   1:  PR[GP1:91,1] = PR[GP1:90,1] + -1.924;
   1:  PR[GP1:91,2] = PR[GP1:90,2] + -33.395;
   1:L PR[91] 10mm/sec CNT100;
   1:  PR[GP1:91,1] = PR[GP1:90,1] + -0.973;
   1:  PR[GP1:91,2] = PR[GP1:90,2] + -33.399;
   1:L PR[91] 10mm/sec CNT100;
   1:  PR[GP1:91,1] = PR[GP1:90,1] + 1.461;
   1:  PR[GP1:91,2] = PR[GP1:90,2] + -33.302;
   1:L PR[91] 10mm/sec CNT100;
   1:  PR[GP1:91,1] = PR[GP1:90,1] + 2.467;
   1:  PR[GP1:91,2] = PR[GP1:90,2] + -33.088;
   1:L PR[91] 10mm/sec CNT100;
   1:  PR[GP1:91,1] = PR[GP1:90,1] + 2.933;
   1:  PR[GP1:91,2] = PR[GP1:90,2] + -33.462;
   1:L PR[91] 10mm/sec CNT100;
   1:  PR[GP1:91,1] = PR[GP1:90,1] + 7.580;
   1:  PR[GP1:91,2] = PR[GP1:90,2] + -34.974;
   1:L PR[91] 10mm/sec CNT100;
   1:  PR[GP1:91,1] = PR[GP1:90,1] + 15.667;
   1:  PR[GP1:91,2] = PR[GP1:90,2] + -37.774;
   1:L PR[91] 10mm/sec CNT100;
   1:  PR[GP1:91,1] = PR[GP1:90,1] + 15.934;
   1:  PR[GP1:91,2] = PR[GP1:90,2] + -37.809;
   1:L PR[91] 10mm/sec CNT100;
   1:  PR[GP1:91,1] = PR[GP1:90,1] + 16.325;
   1:  PR[GP1:91,2] = PR[GP1:90,2] + -37.796;
   1:L PR[91] 10mm/sec CNT100;
   1:  PR[GP1:91,1] = PR[GP1:90,1] + 29.643;
   1:  PR[GP1:91,2] = PR[GP1:90,2] + -37.737;
   1:L PR[91] 10mm/sec CNT100;
   1:  PR[GP1:91,1] = PR[GP1:90,1] + 30.537;
   1:  PR[GP1:91,2] = PR[GP1:90,2] + -37.545;
   1:L PR[91] 10mm/sec CNT100;
   1:  PR[GP1:91,1] = PR[GP1:90,1] + 31.585;
   1:  PR[GP1:91,2] = PR[GP1:90,2] + -37.132;
   1:L PR[91] 10mm/sec CNT100;
   1:  PR[GP1:91,1] = PR[GP1:90,1] + 42.786;
   1:  PR[GP1:91,2] = PR[GP1:90,2] + -33.162;
   1:L PR[91] 10mm/sec CNT100;
   1:  PR[GP1:91,1] = PR[GP1:90,1] + 44.099;
   1:  PR[GP1:91,2] = PR[GP1:90,2] + -32.349;
   1:L PR[91] 10mm/sec CNT100;
   1:  PR[GP1:91,1] = PR[GP1:90,1] + 45.422;
   1:  PR[GP1:91,2] = PR[GP1:90,2] + -31.177;
   1:L PR[91] 10mm/sec CNT100;
   1:  PR[GP1:91,1] = PR[GP1:90,1] + 53.505;
   1:  PR[GP1:91,2] = PR[GP1:90,2] + -24.634;
   1:L PR[91] 10mm/sec CNT100;
   1:  PR[GP1:91,1] = PR[GP1:90,1] + 54.760;
   1:  PR[GP1:91,2] = PR[GP1:90,2] + -23.005;
   1:L PR[91] 10mm/sec CNT100;
   1:  PR[GP1:91,1] = PR[GP1:90,1] + 55.835;
   1:  PR[GP1:91,2] = PR[GP1:90,2] + -20.942;
   1:L PR[91] 10mm/sec CNT100;
   1:  PR[GP1:91,1] = PR[GP1:90,1] + 60.576;
   1:  PR[GP1:91,2] = PR[GP1:90,2] + -13.042;
   1:L PR[91] 10mm/sec CNT100;
   1:  PR[GP1:91,1] = PR[GP1:90,1] + 61.225;
   1:  PR[GP1:91,2] = PR[GP1:90,2] + -10.871;
   1:L PR[91] 10mm/sec CNT100;
   1:  PR[GP1:91,1] = PR[GP1:90,1] + 61.456;
   1:  PR[GP1:91,2] = PR[GP1:90,2] + -8.401;
   1:L PR[91] 10mm/sec CNT100;
   1:  PR[GP1:91,1] = PR[GP1:90,1] + 63.007;
   1:  PR[GP1:91,2] = PR[GP1:90,2] + 0.023;
   1:L PR[91] 10mm/sec CNT100;
   1:  PR[GP1:91,1] = PR[GP1:90,1] + 62.779;
   1:  PR[GP1:91,2] = PR[GP1:90,2] + 2.498;
   1:L PR[91] 10mm/sec CNT100;
   1:  PR[GP1:91,1] = PR[GP1:90,1] + 61.234;
   1:  PR[GP1:91,2] = PR[GP1:90,2] + 10.834;
   1:L PR[91] 10mm/sec CNT100;
   1:  PR[GP1:91,1] = PR[GP1:90,1] + 60.572;
   1:  PR[GP1:91,2] = PR[GP1:90,2] + 13.050;
   1:L PR[91] 10mm/sec CNT100;
   1:  PR[GP1:91,1] = PR[GP1:90,1] + 59.492;
   1:  PR[GP1:91,2] = PR[GP1:90,2] + 15.141;
   1:L PR[91] 10mm/sec CNT100;
   1:  PR[GP1:91,1] = PR[GP1:90,1] + 54.775;
   1:  PR[GP1:91,2] = PR[GP1:90,2] + 22.977;
   1:L PR[91] 10mm/sec CNT100;
   1:  PR[GP1:91,1] = PR[GP1:90,1] + 53.500;
   1:  PR[GP1:91,2] = PR[GP1:90,2] + 24.633;
   1:L PR[91] 10mm/sec CNT100;
   1:  PR[GP1:91,1] = PR[GP1:90,1] + 52.084;
   1:  PR[GP1:91,2] = PR[GP1:90,2] + 25.898;
   1:L PR[91] 10mm/sec CNT100;
   1:  PR[GP1:91,1] = PR[GP1:90,1] + 44.120;
   1:  PR[GP1:91,2] = PR[GP1:90,2] + 32.328;
   1:L PR[91] 10mm/sec CNT100;
   1:  PR[GP1:91,1] = PR[GP1:90,1] + 42.785;
   1:  PR[GP1:91,2] = PR[GP1:90,2] + 33.155;
   1:L PR[91] 10mm/sec CNT100;
   1:  PR[GP1:91,1] = PR[GP1:90,1] + 41.460;
   1:  PR[GP1:91,2] = PR[GP1:90,2] + 33.684;
   1:L PR[91] 10mm/sec CNT100;
   1:  PR[GP1:91,1] = PR[GP1:90,1] + 30.563;
   1:  PR[GP1:91,2] = PR[GP1:90,2] + 37.531;
   1:L PR[91] 10mm/sec CNT100;
   1:  PR[GP1:91,1] = PR[GP1:90,1] + 29.649;
   1:  PR[GP1:91,2] = PR[GP1:90,2] + 37.728;
   1:L PR[91] 10mm/sec CNT100;
   1:  PR[GP1:91,1] = PR[GP1:90,1] + 28.809;
   1:  PR[GP1:91,2] = PR[GP1:90,2] + 37.760;
   1:L PR[91] 10mm/sec CNT100;
   1:  PR[GP1:91,1] = PR[GP1:90,1] + 15.964;
   1:  PR[GP1:91,2] = PR[GP1:90,2] + 37.805;
   1:L PR[91] 10mm/sec CNT100;
   1:  PR[GP1:91,1] = PR[GP1:90,1] + 15.687;
   1:  PR[GP1:91,2] = PR[GP1:90,2] + 37.768;
   1:L PR[91] 10mm/sec CNT100;
   1:  PR[GP1:91,1] = PR[GP1:90,1] + 7.446;
   1:  PR[GP1:91,2] = PR[GP1:90,2] + 34.920;
   1:L PR[91] 10mm/sec CNT100;
   1:  PR[GP1:91,1] = PR[GP1:90,1] + 3.248;
   1:  PR[GP1:91,2] = PR[GP1:90,2] + 33.556;
   1:L PR[91] 10mm/sec CNT100;
   1:  PR[GP1:91,1] = PR[GP1:90,1] + 2.438;
   1:  PR[GP1:91,2] = PR[GP1:90,2] + 33.105;
   1:L PR[91] 10mm/sec CNT100;
   1:  PR[GP1:91,1] = PR[GP1:90,1] + 0.251;
   1:  PR[GP1:91,2] = PR[GP1:90,2] + 33.820;
   1:  PR[GP1:91,3] = PR[GP1:90,3] + 71.820;
   1:L PR[91] 10mm/sec CNT100;
   1:  PR[GP1:91,1] = PR[GP1:90,1] + -1.865;
   1:  PR[GP1:91,2] = PR[GP1:90,2] + 33.807;
   1:L PR[91] 10mm/sec CNT100;
   1:  PR[GP1:91,1] = PR[GP1:90,1] + -14.438;
   1:  PR[GP1:91,2] = PR[GP1:90,2] + 37.919;
   1:L PR[91] 10mm/sec CNT100;
   1:  PR[GP1:91,1] = PR[GP1:90,1] + -28.437;
   1:  PR[GP1:91,2] = PR[GP1:90,2] + 37.848;
   1:L PR[91] 10mm/sec CNT100;
   1:  PR[GP1:91,1] = PR[GP1:90,1] + -28.988;
   1:  PR[GP1:91,2] = PR[GP1:90,2] + 37.729;
   1:L PR[91] 10mm/sec CNT100;
   1:  PR[GP1:91,1] = PR[GP1:90,1] + -29.665;
   1:  PR[GP1:91,2] = PR[GP1:90,2] + 37.461;
   1:L PR[91] 10mm/sec CNT100;
   1:  PR[GP1:91,1] = PR[GP1:90,1] + -41.584;
   1:  PR[GP1:91,2] = PR[GP1:90,2] + 33.229;
   1:L PR[91] 10mm/sec CNT100;
   1:  PR[GP1:91,1] = PR[GP1:90,1] + -42.596;
   1:  PR[GP1:91,2] = PR[GP1:90,2] + 32.598;
   1:L PR[91] 10mm/sec CNT100;
   1:  PR[GP1:91,1] = PR[GP1:90,1] + -43.632;
   1:  PR[GP1:91,2] = PR[GP1:90,2] + 31.678;
   1:L PR[91] 10mm/sec CNT100;
   1:  PR[GP1:91,1] = PR[GP1:90,1] + -52.315;
   1:  PR[GP1:91,2] = PR[GP1:90,2] + 24.651;
   1:L PR[91] 10mm/sec CNT100;
   1:  PR[GP1:91,1] = PR[GP1:90,1] + -53.335;
   1:  PR[GP1:91,2] = PR[GP1:90,2] + 23.323;
   1:L PR[91] 10mm/sec CNT100;
   1:  PR[GP1:91,1] = PR[GP1:90,1] + -54.225;
   1:  PR[GP1:91,2] = PR[GP1:90,2] + 21.596;
   1:L PR[91] 10mm/sec CNT100;
   1:  PR[GP1:91,1] = PR[GP1:90,1] + -59.359;
   1:  PR[GP1:91,2] = PR[GP1:90,2] + 13.022;
   1:L PR[91] 10mm/sec CNT100;
   1:  PR[GP1:91,1] = PR[GP1:90,1] + -59.908;
   1:  PR[GP1:91,2] = PR[GP1:90,2] + 11.157;
   1:L PR[91] 10mm/sec CNT100;
   1:  PR[GP1:91,1] = PR[GP1:90,1] + -60.096;
   1:  PR[GP1:91,2] = PR[GP1:90,2] + 9.107;
   1:L PR[91] 10mm/sec CNT100;
   1:  PR[GP1:91,1] = PR[GP1:90,1] + -61.780;
   1:  PR[GP1:91,2] = PR[GP1:90,2] + -0.032;
   1:L PR[91] 10mm/sec CNT100;
   1:  PR[GP1:91,1] = PR[GP1:90,1] + -61.594;
   1:  PR[GP1:91,2] = PR[GP1:90,2] + -2.098;
   1:L PR[91] 10mm/sec CNT100;
   1:  PR[GP1:91,1] = PR[GP1:90,1] + -59.915;
   1:  PR[GP1:91,2] = PR[GP1:90,2] + -11.142;
   1:L PR[91] 10mm/sec CNT100;
   1:  PR[GP1:91,1] = PR[GP1:90,1] + -59.352;
   1:  PR[GP1:91,2] = PR[GP1:90,2] + -13.053;
   1:L PR[91] 10mm/sec CNT100;
   1:  PR[GP1:91,1] = PR[GP1:90,1] + -58.438;
   1:  PR[GP1:91,2] = PR[GP1:90,2] + -14.845;
   1:L PR[91] 10mm/sec CNT100;
   1:  PR[GP1:91,1] = PR[GP1:90,1] + -53.343;
   1:  PR[GP1:91,2] = PR[GP1:90,2] + -23.322;
   1:L PR[91] 10mm/sec CNT100;
   1:  PR[GP1:91,1] = PR[GP1:90,1] + -52.301;
   1:  PR[GP1:91,2] = PR[GP1:90,2] + -24.678;
   1:L PR[91] 10mm/sec CNT100;
   1:  PR[GP1:91,1] = PR[GP1:90,1] + -51.126;
   1:  PR[GP1:91,2] = PR[GP1:90,2] + -25.732;
   1:L PR[91] 10mm/sec CNT100;
   1:  PR[GP1:91,1] = PR[GP1:90,1] + -42.599;
   1:  PR[GP1:91,2] = PR[GP1:90,2] + -32.605;
   1:L PR[91] 10mm/sec CNT100;
   1:  PR[GP1:91,1] = PR[GP1:90,1] + -41.563;
   1:  PR[GP1:91,2] = PR[GP1:90,2] + -33.250;
   1:L PR[91] 10mm/sec CNT100;
   1:  PR[GP1:91,1] = PR[GP1:90,1] + -40.542;
   1:  PR[GP1:91,2] = PR[GP1:90,2] + -33.660;
   1:L PR[91] 10mm/sec CNT100;
   1:  PR[GP1:91,1] = PR[GP1:90,1] + -28.983;
   1:  PR[GP1:91,2] = PR[GP1:90,2] + -37.738;
   1:L PR[91] 10mm/sec CNT100;
   1:  PR[GP1:91,1] = PR[GP1:90,1] + -28.411;
   1:  PR[GP1:91,2] = PR[GP1:90,2] + -37.862;
   1:L PR[91] 10mm/sec CNT100;
   1:  PR[GP1:91,1] = PR[GP1:90,1] + -27.878;
   1:  PR[GP1:91,2] = PR[GP1:90,2] + -37.882;
   1:L PR[91] 10mm/sec CNT100;
   1:  PR[GP1:91,1] = PR[GP1:90,1] + -14.415;
   1:  PR[GP1:91,2] = PR[GP1:90,2] + -37.925;
   1:L PR[91] 10mm/sec CNT100;
   1:  PR[GP1:91,1] = PR[GP1:90,1] + -1.865;
   1:  PR[GP1:91,2] = PR[GP1:90,2] + -33.819;
   1:L PR[91] 10mm/sec CNT100;
   1:  PR[GP1:91,1] = PR[GP1:90,1] + 0.338;
   1:  PR[GP1:91,2] = PR[GP1:90,2] + -33.830;
   1:L PR[91] 10mm/sec CNT100;
   1:  PR[GP1:91,1] = PR[GP1:90,1] + 1.823;
   1:  PR[GP1:91,2] = PR[GP1:90,2] + -33.770;
   1:L PR[91] 10mm/sec CNT100;
   1:  PR[GP1:91,1] = PR[GP1:90,1] + 2.534;
   1:  PR[GP1:91,2] = PR[GP1:90,2] + -33.619;
   1:L PR[91] 10mm/sec CNT100;
   1:  PR[GP1:91,1] = PR[GP1:90,1] + 2.874;
   1:  PR[GP1:91,2] = PR[GP1:90,2] + -33.893;
   1:L PR[91] 10mm/sec CNT100;
   1:  PR[GP1:91,1] = PR[GP1:90,1] + 14.365;
   1:  PR[GP1:91,2] = PR[GP1:90,2] + -37.631;
   1:L PR[91] 10mm/sec CNT100;
   1:  PR[GP1:91,1] = PR[GP1:90,1] + 15.195;
   1:  PR[GP1:91,2] = PR[GP1:90,2] + -37.918;
   1:L PR[91] 10mm/sec CNT100;
   1:  PR[GP1:91,1] = PR[GP1:90,1] + 29.235;
   1:  PR[GP1:91,2] = PR[GP1:90,2] + -37.861;
   1:L PR[91] 10mm/sec CNT100;
   1:  PR[GP1:91,1] = PR[GP1:90,1] + 29.785;
   1:  PR[GP1:91,2] = PR[GP1:90,2] + -37.742;
   1:L PR[91] 10mm/sec CNT100;
   1:  PR[GP1:91,1] = PR[GP1:90,1] + 30.462;
   1:  PR[GP1:91,2] = PR[GP1:90,2] + -37.476;
   1:L PR[91] 10mm/sec CNT100;
   1:  PR[GP1:91,1] = PR[GP1:90,1] + 42.388;
   1:  PR[GP1:91,2] = PR[GP1:90,2] + -33.249;
   1:L PR[91] 10mm/sec CNT100;
   1:  PR[GP1:91,1] = PR[GP1:90,1] + 43.393;
   1:  PR[GP1:91,2] = PR[GP1:90,2] + -32.626;
   1:L PR[91] 10mm/sec CNT100;
   1:  PR[GP1:91,1] = PR[GP1:90,1] + 44.423;
   1:  PR[GP1:91,2] = PR[GP1:90,2] + -31.714;
   1:L PR[91] 10mm/sec CNT100;
   1:  PR[GP1:91,1] = PR[GP1:90,1] + 53.109;
   1:  PR[GP1:91,2] = PR[GP1:90,2] + -24.683;
   1:L PR[91] 10mm/sec CNT100;
   1:  PR[GP1:91,1] = PR[GP1:90,1] + 54.141;
   1:  PR[GP1:91,2] = PR[GP1:90,2] + -23.343;
   1:L PR[91] 10mm/sec CNT100;
   1:  PR[GP1:91,1] = PR[GP1:90,1] + 55.034;
   1:  PR[GP1:91,2] = PR[GP1:90,2] + -21.630;
   1:L PR[91] 10mm/sec CNT100;
   1:  PR[GP1:91,1] = PR[GP1:90,1] + 60.170;
   1:  PR[GP1:91,2] = PR[GP1:90,2] + -13.073;
   1:L PR[91] 10mm/sec CNT100;
   1:  PR[GP1:91,1] = PR[GP1:90,1] + 60.718;
   1:  PR[GP1:91,2] = PR[GP1:90,2] + -11.237;
   1:L PR[91] 10mm/sec CNT100;
   1:  PR[GP1:91,1] = PR[GP1:90,1] + 60.915;
   1:  PR[GP1:91,2] = PR[GP1:90,2] + -9.131;
   1:L PR[91] 10mm/sec CNT100;
   1:  PR[GP1:91,1] = PR[GP1:90,1] + 62.601;
   1:  PR[GP1:91,2] = PR[GP1:90,2] + 0.023;
   1:L PR[91] 10mm/sec CNT100;
   1:  PR[GP1:91,1] = PR[GP1:90,1] + 62.405;
   1:  PR[GP1:91,2] = PR[GP1:90,2] + 2.148;
   1:L PR[91] 10mm/sec CNT100;
   1:  PR[GP1:91,1] = PR[GP1:90,1] + 60.727;
   1:  PR[GP1:91,2] = PR[GP1:90,2] + 11.199;
   1:L PR[91] 10mm/sec CNT100;
   1:  PR[GP1:91,1] = PR[GP1:90,1] + 60.165;
   1:  PR[GP1:91,2] = PR[GP1:90,2] + 13.080;
   1:L PR[91] 10mm/sec CNT100;
   1:  PR[GP1:91,1] = PR[GP1:90,1] + 59.248;
   1:  PR[GP1:91,2] = PR[GP1:90,2] + 14.857;
   1:L PR[91] 10mm/sec CNT100;
   1:  PR[GP1:91,1] = PR[GP1:90,1] + 54.157;
   1:  PR[GP1:91,2] = PR[GP1:90,2] + 23.314;
   1:L PR[91] 10mm/sec CNT100;
   1:  PR[GP1:91,1] = PR[GP1:90,1] + 53.104;
   1:  PR[GP1:91,2] = PR[GP1:90,2] + 24.681;
   1:L PR[91] 10mm/sec CNT100;
   1:  PR[GP1:91,1] = PR[GP1:90,1] + 51.935;
   1:  PR[GP1:91,2] = PR[GP1:90,2] + 25.727;
   1:L PR[91] 10mm/sec CNT100;
   1:  PR[GP1:91,1] = PR[GP1:90,1] + 43.415;
   1:  PR[GP1:91,2] = PR[GP1:90,2] + 32.604;
   1:L PR[91] 10mm/sec CNT100;
   1:  PR[GP1:91,1] = PR[GP1:90,1] + 42.387;
   1:  PR[GP1:91,2] = PR[GP1:90,2] + 33.241;
   1:L PR[91] 10mm/sec CNT100;
   1:  PR[GP1:91,1] = PR[GP1:90,1] + 41.363;
   1:  PR[GP1:91,2] = PR[GP1:90,2] + 33.650;
   1:L PR[91] 10mm/sec CNT100;
   1:  PR[GP1:91,1] = PR[GP1:90,1] + 29.812;
   1:  PR[GP1:91,2] = PR[GP1:90,2] + 37.728;
   1:L PR[91] 10mm/sec CNT100;
   1:  PR[GP1:91,1] = PR[GP1:90,1] + 29.241;
   1:  PR[GP1:91,2] = PR[GP1:90,2] + 37.851;
   1:L PR[91] 10mm/sec CNT100;
   1:  PR[GP1:91,1] = PR[GP1:90,1] + 28.711;
   1:  PR[GP1:91,2] = PR[GP1:90,2] + 37.871;
   1:L PR[91] 10mm/sec CNT100;
   1:  PR[GP1:91,1] = PR[GP1:90,1] + 15.216;
   1:  PR[GP1:91,2] = PR[GP1:90,2] + 37.913;
   1:L PR[91] 10mm/sec CNT100;
   1:  PR[GP1:91,1] = PR[GP1:90,1] + 14.351;
   1:  PR[GP1:91,2] = PR[GP1:90,2] + 37.614;
   1:L PR[91] 10mm/sec CNT100;
   1:  PR[GP1:91,1] = PR[GP1:90,1] + 3.055;
   1:  PR[GP1:91,2] = PR[GP1:90,2] + 33.942;
   1:L PR[91] 10mm/sec CNT100;
   1:  PR[GP1:91,1] = PR[GP1:90,1] + 2.503;
   1:  PR[GP1:91,2] = PR[GP1:90,2] + 33.635;
   1:L PR[91] 10mm/sec CNT100;
   1:  PR[GP1:91,1] = PR[GP1:90,1] + 1.540;
   1:  PR[GP1:91,2] = PR[GP1:90,2] + 34.250;
   1:  PR[GP1:91,3] = PR[GP1:90,3] + 73.150;
   1:L PR[91] 10mm/sec CNT100;
   1:  PR[GP1:91,1] = PR[GP1:90,1] + -1.806;
   1:  PR[GP1:91,2] = PR[GP1:90,2] + 34.230;
   1:L PR[91] 10mm/sec CNT100;
   1:  PR[GP1:91,1] = PR[GP1:90,1] + -12.018;
   1:  PR[GP1:91,2] = PR[GP1:90,2] + 37.561;
   1:L PR[91] 10mm/sec CNT100;
   1:  PR[GP1:91,1] = PR[GP1:90,1] + -13.780;
   1:  PR[GP1:91,2] = PR[GP1:90,2] + 38.106;
   1:L PR[91] 10mm/sec CNT100;
   1:  PR[GP1:91,1] = PR[GP1:90,1] + -14.321;
   1:  PR[GP1:91,2] = PR[GP1:90,2] + 38.125;
   1:L PR[91] 10mm/sec CNT100;
   1:  PR[GP1:91,1] = PR[GP1:90,1] + -20.781;
   1:  PR[GP1:91,2] = PR[GP1:90,2] + 38.007;
   1:L PR[91] 10mm/sec CNT100;
   1:  PR[GP1:91,1] = PR[GP1:90,1] + -28.027;
   1:  PR[GP1:91,2] = PR[GP1:90,2] + 37.971;
   1:L PR[91] 10mm/sec CNT100;
   1:  PR[GP1:91,1] = PR[GP1:90,1] + -28.235;
   1:  PR[GP1:91,2] = PR[GP1:90,2] + 37.926;
   1:L PR[91] 10mm/sec CNT100;
   1:  PR[GP1:91,1] = PR[GP1:90,1] + -28.540;
   1:  PR[GP1:91,2] = PR[GP1:90,2] + 37.805;
   1:L PR[91] 10mm/sec CNT100;
   1:  PR[GP1:91,1] = PR[GP1:90,1] + -41.184;
   1:  PR[GP1:91,2] = PR[GP1:90,2] + 33.316;
   1:L PR[91] 10mm/sec CNT100;
   1:  PR[GP1:91,1] = PR[GP1:90,1] + -41.888;
   1:  PR[GP1:91,2] = PR[GP1:90,2] + 32.877;
   1:L PR[91] 10mm/sec CNT100;
   1:  PR[GP1:91,1] = PR[GP1:90,1] + -42.628;
   1:  PR[GP1:91,2] = PR[GP1:90,2] + 32.220;
   1:L PR[91] 10mm/sec CNT100;
   1:  PR[GP1:91,1] = PR[GP1:90,1] + -51.915;
   1:  PR[GP1:91,2] = PR[GP1:90,2] + 24.704;
   1:L PR[91] 10mm/sec CNT100;
   1:  PR[GP1:91,1] = PR[GP1:90,1] + -52.715;
   1:  PR[GP1:91,2] = PR[GP1:90,2] + 23.663;
   1:L PR[91] 10mm/sec CNT100;
   1:  PR[GP1:91,1] = PR[GP1:90,1] + -53.423;
   1:  PR[GP1:91,2] = PR[GP1:90,2] + 22.290;
   1:L PR[91] 10mm/sec CNT100;
   1:  PR[GP1:91,1] = PR[GP1:90,1] + -58.951;
   1:  PR[GP1:91,2] = PR[GP1:90,2] + 13.056;
   1:L PR[91] 10mm/sec CNT100;
   1:  PR[GP1:91,1] = PR[GP1:90,1] + -59.400;
   1:  PR[GP1:91,2] = PR[GP1:90,2] + 11.531;
   1:L PR[91] 10mm/sec CNT100;
   1:  PR[GP1:91,1] = PR[GP1:90,1] + -59.555;
   1:  PR[GP1:91,2] = PR[GP1:90,2] + 9.836;
   1:L PR[91] 10mm/sec CNT100;
   1:  PR[GP1:91,1] = PR[GP1:90,1] + -61.374;
   1:  PR[GP1:91,2] = PR[GP1:90,2] + -0.032;
   1:L PR[91] 10mm/sec CNT100;
   1:  PR[GP1:91,1] = PR[GP1:90,1] + -61.218;
   1:  PR[GP1:91,2] = PR[GP1:90,2] + -1.757;
   1:L PR[91] 10mm/sec CNT100;
   1:  PR[GP1:91,1] = PR[GP1:90,1] + -59.407;
   1:  PR[GP1:91,2] = PR[GP1:90,2] + -11.516;
   1:L PR[91] 10mm/sec CNT100;
   1:  PR[GP1:91,1] = PR[GP1:90,1] + -58.944;
   1:  PR[GP1:91,2] = PR[GP1:90,2] + -13.087;
   1:L PR[91] 10mm/sec CNT100;
   1:  PR[GP1:91,1] = PR[GP1:90,1] + -58.191;
   1:  PR[GP1:91,2] = PR[GP1:90,2] + -14.562;
   1:L PR[91] 10mm/sec CNT100;
   1:  PR[GP1:91,1] = PR[GP1:90,1] + -52.722;
   1:  PR[GP1:91,2] = PR[GP1:90,2] + -23.662;
   1:L PR[91] 10mm/sec CNT100;
   1:  PR[GP1:91,1] = PR[GP1:90,1] + -51.901;
   1:  PR[GP1:91,2] = PR[GP1:90,2] + -24.731;
   1:L PR[91] 10mm/sec CNT100;
   1:  PR[GP1:91,1] = PR[GP1:90,1] + -50.973;
   1:  PR[GP1:91,2] = PR[GP1:90,2] + -25.564;
   1:L PR[91] 10mm/sec CNT100;
   1:  PR[GP1:91,1] = PR[GP1:90,1] + -41.890;
   1:  PR[GP1:91,2] = PR[GP1:90,2] + -32.884;
   1:L PR[91] 10mm/sec CNT100;
   1:  PR[GP1:91,1] = PR[GP1:90,1] + -41.163;
   1:  PR[GP1:91,2] = PR[GP1:90,2] + -33.337;
   1:L PR[91] 10mm/sec CNT100;
   1:  PR[GP1:91,1] = PR[GP1:90,1] + -40.442;
   1:  PR[GP1:91,2] = PR[GP1:90,2] + -33.627;
   1:L PR[91] 10mm/sec CNT100;
   1:  PR[GP1:91,1] = PR[GP1:90,1] + -28.228;
   1:  PR[GP1:91,2] = PR[GP1:90,2] + -37.936;
   1:L PR[91] 10mm/sec CNT100;
   1:  PR[GP1:91,1] = PR[GP1:90,1] + -28.000;
   1:  PR[GP1:91,2] = PR[GP1:90,2] + -37.985;
   1:L PR[91] 10mm/sec CNT100;
   1:  PR[GP1:91,1] = PR[GP1:90,1] + -27.778;
   1:  PR[GP1:91,2] = PR[GP1:90,2] + -37.994;
   1:L PR[91] 10mm/sec CNT100;
   1:  PR[GP1:91,1] = PR[GP1:90,1] + -20.782;
   1:  PR[GP1:91,2] = PR[GP1:90,2] + -38.016;
   1:L PR[91] 10mm/sec CNT100;
   1:  PR[GP1:91,1] = PR[GP1:90,1] + -14.301;
   1:  PR[GP1:91,2] = PR[GP1:90,2] + -38.131;
   1:L PR[91] 10mm/sec CNT100;
   1:  PR[GP1:91,1] = PR[GP1:90,1] + -13.759;
   1:  PR[GP1:91,2] = PR[GP1:90,2] + -38.111;
   1:L PR[91] 10mm/sec CNT100;
   1:  PR[GP1:91,1] = PR[GP1:90,1] + -11.599;
   1:  PR[GP1:91,2] = PR[GP1:90,2] + -37.439;
   1:L PR[91] 10mm/sec CNT100;
   1:  PR[GP1:91,1] = PR[GP1:90,1] + -1.806;
   1:  PR[GP1:91,2] = PR[GP1:90,2] + -34.243;
   1:L PR[91] 10mm/sec CNT100;
   1:  PR[GP1:91,1] = PR[GP1:90,1] + 1.649;
   1:  PR[GP1:91,2] = PR[GP1:90,2] + -34.260;
   1:L PR[91] 10mm/sec CNT100;
   1:  PR[GP1:91,1] = PR[GP1:90,1] + 2.184;
   1:  PR[GP1:91,2] = PR[GP1:90,2] + -34.238;
   1:L PR[91] 10mm/sec CNT100;
   1:  PR[GP1:91,1] = PR[GP1:90,1] + 2.600;
   1:  PR[GP1:91,2] = PR[GP1:90,2] + -34.150;
   1:L PR[91] 10mm/sec CNT100;
   1:  PR[GP1:91,1] = PR[GP1:90,1] + 2.815;
   1:  PR[GP1:91,2] = PR[GP1:90,2] + -34.323;
   1:L PR[91] 10mm/sec CNT100;
   1:  PR[GP1:91,1] = PR[GP1:90,1] + 7.942;
   1:  PR[GP1:91,2] = PR[GP1:90,2] + -35.991;
   1:L PR[91] 10mm/sec CNT100;
   1:  PR[GP1:91,1] = PR[GP1:90,1] + 12.414;
   1:  PR[GP1:91,2] = PR[GP1:90,2] + -37.437;
   1:L PR[91] 10mm/sec CNT100;
   1:  PR[GP1:91,1] = PR[GP1:90,1] + 14.577;
   1:  PR[GP1:91,2] = PR[GP1:90,2] + -38.111;
   1:L PR[91] 10mm/sec CNT100;
   1:  PR[GP1:91,1] = PR[GP1:90,1] + 15.119;
   1:  PR[GP1:91,2] = PR[GP1:90,2] + -38.130;
   1:L PR[91] 10mm/sec CNT100;
   1:  PR[GP1:91,1] = PR[GP1:90,1] + 21.601;
   1:  PR[GP1:91,2] = PR[GP1:90,2] + -38.016;
   1:L PR[91] 10mm/sec CNT100;
   1:  PR[GP1:91,1] = PR[GP1:90,1] + 28.827;
   1:  PR[GP1:91,2] = PR[GP1:90,2] + -37.984;
   1:L PR[91] 10mm/sec CNT100;
   1:  PR[GP1:91,1] = PR[GP1:90,1] + 29.033;
   1:  PR[GP1:91,2] = PR[GP1:90,2] + -37.940;
   1:L PR[91] 10mm/sec CNT100;
   1:  PR[GP1:91,1] = PR[GP1:90,1] + 29.338;
   1:  PR[GP1:91,2] = PR[GP1:90,2] + -37.819;
   1:L PR[91] 10mm/sec CNT100;
   1:  PR[GP1:91,1] = PR[GP1:90,1] + 41.989;
   1:  PR[GP1:91,2] = PR[GP1:90,2] + -33.336;
   1:L PR[91] 10mm/sec CNT100;
   1:  PR[GP1:91,1] = PR[GP1:90,1] + 42.688;
   1:  PR[GP1:91,2] = PR[GP1:90,2] + -32.903;
   1:L PR[91] 10mm/sec CNT100;
   1:  PR[GP1:91,1] = PR[GP1:90,1] + 43.423;
   1:  PR[GP1:91,2] = PR[GP1:90,2] + -32.251;
   1:L PR[91] 10mm/sec CNT100;
   1:  PR[GP1:91,1] = PR[GP1:90,1] + 52.713;
   1:  PR[GP1:91,2] = PR[GP1:90,2] + -24.731;
   1:L PR[91] 10mm/sec CNT100;
   1:  PR[GP1:91,1] = PR[GP1:90,1] + 53.522;
   1:  PR[GP1:91,2] = PR[GP1:90,2] + -23.681;
   1:L PR[91] 10mm/sec CNT100;
   1:  PR[GP1:91,1] = PR[GP1:90,1] + 54.232;
   1:  PR[GP1:91,2] = PR[GP1:90,2] + -22.319;
   1:L PR[91] 10mm/sec CNT100;
   1:  PR[GP1:91,1] = PR[GP1:90,1] + 59.763;
   1:  PR[GP1:91,2] = PR[GP1:90,2] + -13.103;
   1:L PR[91] 10mm/sec CNT100;
   1:  PR[GP1:91,1] = PR[GP1:90,1] + 60.212;
   1:  PR[GP1:91,2] = PR[GP1:90,2] + -11.602;
   1:L PR[91] 10mm/sec CNT100;
   1:  PR[GP1:91,1] = PR[GP1:90,1] + 60.375;
   1:  PR[GP1:91,2] = PR[GP1:90,2] + -9.861;
   1:L PR[91] 10mm/sec CNT100;
   1:  PR[GP1:91,1] = PR[GP1:90,1] + 62.195;
   1:  PR[GP1:91,2] = PR[GP1:90,2] + 0.023;
   1:L PR[91] 10mm/sec CNT100;
   1:  PR[GP1:91,1] = PR[GP1:90,1] + 62.031;
   1:  PR[GP1:91,2] = PR[GP1:90,2] + 1.798;
   1:L PR[91] 10mm/sec CNT100;
   1:  PR[GP1:91,1] = PR[GP1:90,1] + 60.221;
   1:  PR[GP1:91,2] = PR[GP1:90,2] + 11.564;
   1:L PR[91] 10mm/sec CNT100;
   1:  PR[GP1:91,1] = PR[GP1:90,1] + 59.759;
   1:  PR[GP1:91,2] = PR[GP1:90,2] + 13.110;
   1:L PR[91] 10mm/sec CNT100;
   1:  PR[GP1:91,1] = PR[GP1:90,1] + 59.004;
   1:  PR[GP1:91,2] = PR[GP1:90,2] + 14.573;
   1:L PR[91] 10mm/sec CNT100;
   1:  PR[GP1:91,1] = PR[GP1:90,1] + 53.538;
   1:  PR[GP1:91,2] = PR[GP1:90,2] + 23.652;
   1:L PR[91] 10mm/sec CNT100;
   1:  PR[GP1:91,1] = PR[GP1:90,1] + 52.709;
   1:  PR[GP1:91,2] = PR[GP1:90,2] + 24.729;
   1:L PR[91] 10mm/sec CNT100;
   1:  PR[GP1:91,1] = PR[GP1:90,1] + 51.785;
   1:  PR[GP1:91,2] = PR[GP1:90,2] + 25.555;
   1:L PR[91] 10mm/sec CNT100;
   1:  PR[GP1:91,1] = PR[GP1:90,1] + 42.710;
   1:  PR[GP1:91,2] = PR[GP1:90,2] + 32.881;
   1:L PR[91] 10mm/sec CNT100;
   1:  PR[GP1:91,1] = PR[GP1:90,1] + 41.988;
   1:  PR[GP1:91,2] = PR[GP1:90,2] + 33.328;
   1:L PR[91] 10mm/sec CNT100;
   1:  PR[GP1:91,1] = PR[GP1:90,1] + 41.266;
   1:  PR[GP1:91,2] = PR[GP1:90,2] + 33.616;
   1:L PR[91] 10mm/sec CNT100;
   1:  PR[GP1:91,1] = PR[GP1:90,1] + 29.061;
   1:  PR[GP1:91,2] = PR[GP1:90,2] + 37.925;
   1:L PR[91] 10mm/sec CNT100;
   1:  PR[GP1:91,1] = PR[GP1:90,1] + 28.843;
   1:  PR[GP1:91,2] = PR[GP1:90,2] + 37.972;
   1:L PR[91] 10mm/sec CNT100;
   1:  PR[GP1:91,1] = PR[GP1:90,1] + 21.601;
   1:  PR[GP1:91,2] = PR[GP1:90,2] + 38.007;
   1:L PR[91] 10mm/sec CNT100;
   1:  PR[GP1:91,1] = PR[GP1:90,1] + 15.138;
   1:  PR[GP1:91,2] = PR[GP1:90,2] + 38.124;
   1:L PR[91] 10mm/sec CNT100;
   1:  PR[GP1:91,1] = PR[GP1:90,1] + 14.597;
   1:  PR[GP1:91,2] = PR[GP1:90,2] + 38.105;
   1:L PR[91] 10mm/sec CNT100;
   1:  PR[GP1:91,1] = PR[GP1:90,1] + 12.833;
   1:  PR[GP1:91,2] = PR[GP1:90,2] + 37.560;
   1:L PR[91] 10mm/sec CNT100;
   1:  PR[GP1:91,1] = PR[GP1:90,1] + 2.861;
   1:  PR[GP1:91,2] = PR[GP1:90,2] + 34.328;
   1:L PR[91] 10mm/sec CNT100;
   1:  PR[GP1:91,1] = PR[GP1:90,1] + 2.569;
   1:  PR[GP1:91,2] = PR[GP1:90,2] + 34.166;
   1:L PR[91] 10mm/sec CNT100;
   1:  PR[GP1:91,1] = PR[GP1:90,1] + -1.747;
   1:  PR[GP1:91,2] = PR[GP1:90,2] + 34.652;
   1:  PR[GP1:91,3] = PR[GP1:90,3] + 74.480;
   1:L PR[91] 10mm/sec CNT100;
   1:  PR[GP1:91,1] = PR[GP1:90,1] + -9.248;
   1:  PR[GP1:91,2] = PR[GP1:90,2] + 37.099;
   1:L PR[91] 10mm/sec CNT100;
   1:  PR[GP1:91,1] = PR[GP1:90,1] + -13.132;
   1:  PR[GP1:91,2] = PR[GP1:90,2] + 38.299;
   1:L PR[91] 10mm/sec CNT100;
   1:  PR[GP1:91,1] = PR[GP1:90,1] + -14.404;
   1:  PR[GP1:91,2] = PR[GP1:90,2] + 38.345;
   1:L PR[91] 10mm/sec CNT100;
   1:  PR[GP1:91,1] = PR[GP1:90,1] + -27.562;
   1:  PR[GP1:91,2] = PR[GP1:90,2] + 38.105;
   1:L PR[91] 10mm/sec CNT100;
   1:  PR[GP1:91,1] = PR[GP1:90,1] + -40.783;
   1:  PR[GP1:91,2] = PR[GP1:90,2] + 33.403;
   1:L PR[91] 10mm/sec CNT100;
   1:  PR[GP1:91,1] = PR[GP1:90,1] + -41.179;
   1:  PR[GP1:91,2] = PR[GP1:90,2] + 33.157;
   1:L PR[91] 10mm/sec CNT100;
   1:  PR[GP1:91,1] = PR[GP1:90,1] + -41.625;
   1:  PR[GP1:91,2] = PR[GP1:90,2] + 32.761;
   1:L PR[91] 10mm/sec CNT100;
   1:  PR[GP1:91,1] = PR[GP1:90,1] + -51.515;
   1:  PR[GP1:91,2] = PR[GP1:90,2] + 24.757;
   1:L PR[91] 10mm/sec CNT100;
   1:  PR[GP1:91,1] = PR[GP1:90,1] + -52.094;
   1:  PR[GP1:91,2] = PR[GP1:90,2] + 24.003;
   1:L PR[91] 10mm/sec CNT100;
   1:  PR[GP1:91,1] = PR[GP1:90,1] + -52.620;
   1:  PR[GP1:91,2] = PR[GP1:90,2] + 22.984;
   1:L PR[91] 10mm/sec CNT100;
   1:  PR[GP1:91,1] = PR[GP1:90,1] + -58.543;
   1:  PR[GP1:91,2] = PR[GP1:90,2] + 13.090;
   1:L PR[91] 10mm/sec CNT100;
   1:  PR[GP1:91,1] = PR[GP1:90,1] + -58.892;
   1:  PR[GP1:91,2] = PR[GP1:90,2] + 11.905;
   1:L PR[91] 10mm/sec CNT100;
   1:  PR[GP1:91,1] = PR[GP1:90,1] + -59.015;
   1:  PR[GP1:91,2] = PR[GP1:90,2] + 10.565;
   1:L PR[91] 10mm/sec CNT100;
   1:  PR[GP1:91,1] = PR[GP1:90,1] + -60.968;
   1:  PR[GP1:91,2] = PR[GP1:90,2] + -0.032;
   1:L PR[91] 10mm/sec CNT100;
   1:  PR[GP1:91,1] = PR[GP1:90,1] + -60.843;
   1:  PR[GP1:91,2] = PR[GP1:90,2] + -1.416;
   1:L PR[91] 10mm/sec CNT100;
   1:  PR[GP1:91,1] = PR[GP1:90,1] + -58.899;
   1:  PR[GP1:91,2] = PR[GP1:90,2] + -11.891;
   1:L PR[91] 10mm/sec CNT100;
   1:  PR[GP1:91,1] = PR[GP1:90,1] + -58.536;
   1:  PR[GP1:91,2] = PR[GP1:90,2] + -13.122;
   1:L PR[91] 10mm/sec CNT100;
   1:  PR[GP1:91,1] = PR[GP1:90,1] + -57.945;
   1:  PR[GP1:91,2] = PR[GP1:90,2] + -14.279;
   1:L PR[91] 10mm/sec CNT100;
   1:  PR[GP1:91,1] = PR[GP1:90,1] + -52.101;
   1:  PR[GP1:91,2] = PR[GP1:90,2] + -24.002;
   1:L PR[91] 10mm/sec CNT100;
   1:  PR[GP1:91,1] = PR[GP1:90,1] + -51.501;
   1:  PR[GP1:91,2] = PR[GP1:90,2] + -24.784;
   1:L PR[91] 10mm/sec CNT100;
   1:  PR[GP1:91,1] = PR[GP1:90,1] + -50.820;
   1:  PR[GP1:91,2] = PR[GP1:90,2] + -25.395;
   1:L PR[91] 10mm/sec CNT100;
   1:  PR[GP1:91,1] = PR[GP1:90,1] + -41.180;
   1:  PR[GP1:91,2] = PR[GP1:90,2] + -33.164;
   1:L PR[91] 10mm/sec CNT100;
   1:  PR[GP1:91,1] = PR[GP1:90,1] + -40.762;
   1:  PR[GP1:91,2] = PR[GP1:90,2] + -33.425;
   1:L PR[91] 10mm/sec CNT100;
   1:  PR[GP1:91,1] = PR[GP1:90,1] + -40.342;
   1:  PR[GP1:91,2] = PR[GP1:90,2] + -33.594;
   1:L PR[91] 10mm/sec CNT100;
   1:  PR[GP1:91,1] = PR[GP1:90,1] + -27.544;
   1:  PR[GP1:91,2] = PR[GP1:90,2] + -38.117;
   1:L PR[91] 10mm/sec CNT100;
   1:  PR[GP1:91,1] = PR[GP1:90,1] + -14.387;
   1:  PR[GP1:91,2] = PR[GP1:90,2] + -38.350;
   1:L PR[91] 10mm/sec CNT100;
   1:  PR[GP1:91,1] = PR[GP1:90,1] + -13.086;
   1:  PR[GP1:91,2] = PR[GP1:90,2] + -38.298;
   1:L PR[91] 10mm/sec CNT100;
   1:  PR[GP1:91,1] = PR[GP1:90,1] + -8.382;
   1:  PR[GP1:91,2] = PR[GP1:90,2] + -36.832;
   1:L PR[91] 10mm/sec CNT100;
   1:  PR[GP1:91,1] = PR[GP1:90,1] + -1.748;
   1:  PR[GP1:91,2] = PR[GP1:90,2] + -34.667;
   1:L PR[91] 10mm/sec CNT100;
   1:  PR[GP1:91,1] = PR[GP1:90,1] + 0.835;
   1:  PR[GP1:91,2] = PR[GP1:90,2] + -34.666;
   1:L PR[91] 10mm/sec CNT100;
   1:  PR[GP1:91,1] = PR[GP1:90,1] + 2.564;
   1:  PR[GP1:91,2] = PR[GP1:90,2] + -34.685;
   1:L PR[91] 10mm/sec CNT100;
   1:  PR[GP1:91,1] = PR[GP1:90,1] + 9.196;
   1:  PR[GP1:91,2] = PR[GP1:90,2] + -36.830;
   1:L PR[91] 10mm/sec CNT100;
   1:  PR[GP1:91,1] = PR[GP1:90,1] + 13.930;
   1:  PR[GP1:91,2] = PR[GP1:90,2] + -38.304;
   1:L PR[91] 10mm/sec CNT100;
   1:  PR[GP1:91,1] = PR[GP1:90,1] + 15.203;
   1:  PR[GP1:91,2] = PR[GP1:90,2] + -38.350;
   1:L PR[91] 10mm/sec CNT100;
   1:  PR[GP1:91,1] = PR[GP1:90,1] + 28.362;
   1:  PR[GP1:91,2] = PR[GP1:90,2] + -38.118;
   1:L PR[91] 10mm/sec CNT100;
   1:  PR[GP1:91,1] = PR[GP1:90,1] + 41.590;
   1:  PR[GP1:91,2] = PR[GP1:90,2] + -33.423;
   1:L PR[91] 10mm/sec CNT100;
   1:  PR[GP1:91,1] = PR[GP1:90,1] + 41.982;
   1:  PR[GP1:91,2] = PR[GP1:90,2] + -33.179;
   1:L PR[91] 10mm/sec CNT100;
   1:  PR[GP1:91,1] = PR[GP1:90,1] + 42.424;
   1:  PR[GP1:91,2] = PR[GP1:90,2] + -32.788;
   1:L PR[91] 10mm/sec CNT100;
   1:  PR[GP1:91,1] = PR[GP1:90,1] + 52.317;
   1:  PR[GP1:91,2] = PR[GP1:90,2] + -24.780;
   1:L PR[91] 10mm/sec CNT100;
   1:  PR[GP1:91,1] = PR[GP1:90,1] + 52.904;
   1:  PR[GP1:91,2] = PR[GP1:90,2] + -24.018;
   1:L PR[91] 10mm/sec CNT100;
   1:  PR[GP1:91,1] = PR[GP1:90,1] + 53.431;
   1:  PR[GP1:91,2] = PR[GP1:90,2] + -23.007;
   1:L PR[91] 10mm/sec CNT100;
   1:  PR[GP1:91,1] = PR[GP1:90,1] + 59.357;
   1:  PR[GP1:91,2] = PR[GP1:90,2] + -13.134;
   1:L PR[91] 10mm/sec CNT100;
   1:  PR[GP1:91,1] = PR[GP1:90,1] + 59.705;
   1:  PR[GP1:91,2] = PR[GP1:90,2] + -11.968;
   1:L PR[91] 10mm/sec CNT100;
   1:  PR[GP1:91,1] = PR[GP1:90,1] + 59.834;
   1:  PR[GP1:91,2] = PR[GP1:90,2] + -10.591;
   1:L PR[91] 10mm/sec CNT100;
   1:  PR[GP1:91,1] = PR[GP1:90,1] + 61.789;
   1:  PR[GP1:91,2] = PR[GP1:90,2] + 0.023;
   1:L PR[91] 10mm/sec CNT100;
   1:  PR[GP1:91,1] = PR[GP1:90,1] + 61.657;
   1:  PR[GP1:91,2] = PR[GP1:90,2] + 1.447;
   1:L PR[91] 10mm/sec CNT100;
   1:  PR[GP1:91,1] = PR[GP1:90,1] + 59.714;
   1:  PR[GP1:91,2] = PR[GP1:90,2] + 11.930;
   1:L PR[91] 10mm/sec CNT100;
   1:  PR[GP1:91,1] = PR[GP1:90,1] + 59.353;
   1:  PR[GP1:91,2] = PR[GP1:90,2] + 13.140;
   1:L PR[91] 10mm/sec CNT100;
   1:  PR[GP1:91,1] = PR[GP1:90,1] + 58.760;
   1:  PR[GP1:91,2] = PR[GP1:90,2] + 14.289;
   1:L PR[91] 10mm/sec CNT100;
   1:  PR[GP1:91,1] = PR[GP1:90,1] + 52.920;
   1:  PR[GP1:91,2] = PR[GP1:90,2] + 23.989;
   1:L PR[91] 10mm/sec CNT100;
   1:  PR[GP1:91,1] = PR[GP1:90,1] + 52.313;
   1:  PR[GP1:91,2] = PR[GP1:90,2] + 24.777;
   1:L PR[91] 10mm/sec CNT100;
   1:  PR[GP1:91,1] = PR[GP1:90,1] + 51.635;
   1:  PR[GP1:91,2] = PR[GP1:90,2] + 25.383;
   1:L PR[91] 10mm/sec CNT100;
   1:  PR[GP1:91,1] = PR[GP1:90,1] + 42.005;
   1:  PR[GP1:91,2] = PR[GP1:90,2] + 33.157;
   1:L PR[91] 10mm/sec CNT100;
   1:  PR[GP1:91,1] = PR[GP1:90,1] + 41.590;
   1:  PR[GP1:91,2] = PR[GP1:90,2] + 33.414;
   1:L PR[91] 10mm/sec CNT100;
   1:  PR[GP1:91,1] = PR[GP1:90,1] + 41.168;
   1:  PR[GP1:91,2] = PR[GP1:90,2] + 33.583;
   1:L PR[91] 10mm/sec CNT100;
   1:  PR[GP1:91,1] = PR[GP1:90,1] + 28.380;
   1:  PR[GP1:91,2] = PR[GP1:90,2] + 38.105;
   1:L PR[91] 10mm/sec CNT100;
   1:  PR[GP1:91,1] = PR[GP1:90,1] + 15.222;
   1:  PR[GP1:91,2] = PR[GP1:90,2] + 38.344;
   1:L PR[91] 10mm/sec CNT100;
   1:  PR[GP1:91,1] = PR[GP1:90,1] + 13.949;
   1:  PR[GP1:91,2] = PR[GP1:90,2] + 38.298;
   1:L PR[91] 10mm/sec CNT100;
   1:  PR[GP1:91,1] = PR[GP1:90,1] + 10.062;
   1:  PR[GP1:91,2] = PR[GP1:90,2] + 37.097;
   1:L PR[91] 10mm/sec CNT100;
   1:  PR[GP1:91,1] = PR[GP1:90,1] + 2.563;
   1:  PR[GP1:91,2] = PR[GP1:90,2] + 34.676;
   1:L PR[91] 10mm/sec CNT100;
   1:  PR[GP1:91,1] = PR[GP1:90,1] + -1.689;
   1:  PR[GP1:91,2] = PR[GP1:90,2] + 35.074;
   1:  PR[GP1:91,3] = PR[GP1:90,3] + 75.810;
   1:L PR[91] 10mm/sec CNT100;
   1:  PR[GP1:91,1] = PR[GP1:90,1] + -6.478;
   1:  PR[GP1:91,2] = PR[GP1:90,2] + 36.637;
   1:L PR[91] 10mm/sec CNT100;
   1:  PR[GP1:91,1] = PR[GP1:90,1] + -12.483;
   1:  PR[GP1:91,2] = PR[GP1:90,2] + 38.492;
   1:L PR[91] 10mm/sec CNT100;
   1:  PR[GP1:91,1] = PR[GP1:90,1] + -14.488;
   1:  PR[GP1:91,2] = PR[GP1:90,2] + 38.564;
   1:L PR[91] 10mm/sec CNT100;
   1:  PR[GP1:91,1] = PR[GP1:90,1] + -27.000;
   1:  PR[GP1:91,2] = PR[GP1:90,2] + 38.336;
   1:L PR[91] 10mm/sec CNT100;
   1:  PR[GP1:91,1] = PR[GP1:90,1] + -27.680;
   1:  PR[GP1:91,2] = PR[GP1:90,2] + 38.113;
   1:L PR[91] 10mm/sec CNT100;
   1:  PR[GP1:91,1] = PR[GP1:90,1] + -35.661;
   1:  PR[GP1:91,2] = PR[GP1:90,2] + 35.167;
   1:L PR[91] 10mm/sec CNT100;
   1:  PR[GP1:91,1] = PR[GP1:90,1] + -40.384;
   1:  PR[GP1:91,2] = PR[GP1:90,2] + 33.490;
   1:L PR[91] 10mm/sec CNT100;
   1:  PR[GP1:91,1] = PR[GP1:90,1] + -40.471;
   1:  PR[GP1:91,2] = PR[GP1:90,2] + 33.436;
   1:L PR[91] 10mm/sec CNT100;
   1:  PR[GP1:91,1] = PR[GP1:90,1] + -40.621;
   1:  PR[GP1:91,2] = PR[GP1:90,2] + 33.303;
   1:L PR[91] 10mm/sec CNT100;
   1:  PR[GP1:91,1] = PR[GP1:90,1] + -51.115;
   1:  PR[GP1:91,2] = PR[GP1:90,2] + 24.810;
   1:L PR[91] 10mm/sec CNT100;
   1:  PR[GP1:91,1] = PR[GP1:90,1] + -51.474;
   1:  PR[GP1:91,2] = PR[GP1:90,2] + 24.343;
   1:L PR[91] 10mm/sec CNT100;
   1:  PR[GP1:91,1] = PR[GP1:90,1] + -51.817;
   1:  PR[GP1:91,2] = PR[GP1:90,2] + 23.677;
   1:L PR[91] 10mm/sec CNT100;
   1:  PR[GP1:91,1] = PR[GP1:90,1] + -58.135;
   1:  PR[GP1:91,2] = PR[GP1:90,2] + 13.124;
   1:L PR[91] 10mm/sec CNT100;
   1:  PR[GP1:91,1] = PR[GP1:90,1] + -58.384;
   1:  PR[GP1:91,2] = PR[GP1:90,2] + 12.280;
   1:L PR[91] 10mm/sec CNT100;
   1:  PR[GP1:91,1] = PR[GP1:90,1] + -58.474;
   1:  PR[GP1:91,2] = PR[GP1:90,2] + 11.295;
   1:L PR[91] 10mm/sec CNT100;
   1:  PR[GP1:91,1] = PR[GP1:90,1] + -60.562;
   1:  PR[GP1:91,2] = PR[GP1:90,2] + -0.032;
   1:L PR[91] 10mm/sec CNT100;
   1:  PR[GP1:91,1] = PR[GP1:90,1] + -60.468;
   1:  PR[GP1:91,2] = PR[GP1:90,2] + -1.075;
   1:L PR[91] 10mm/sec CNT100;
   1:  PR[GP1:91,1] = PR[GP1:90,1] + -58.390;
   1:  PR[GP1:91,2] = PR[GP1:90,2] + -12.265;
   1:L PR[91] 10mm/sec CNT100;
   1:  PR[GP1:91,1] = PR[GP1:90,1] + -58.128;
   1:  PR[GP1:91,2] = PR[GP1:90,2] + -13.156;
   1:L PR[91] 10mm/sec CNT100;
   1:  PR[GP1:91,1] = PR[GP1:90,1] + -57.699;
   1:  PR[GP1:91,2] = PR[GP1:90,2] + -13.996;
   1:L PR[91] 10mm/sec CNT100;
   1:  PR[GP1:91,1] = PR[GP1:90,1] + -51.481;
   1:  PR[GP1:91,2] = PR[GP1:90,2] + -24.343;
   1:L PR[91] 10mm/sec CNT100;
   1:  PR[GP1:91,1] = PR[GP1:90,1] + -51.101;
   1:  PR[GP1:91,2] = PR[GP1:90,2] + -24.837;
   1:L PR[91] 10mm/sec CNT100;
   1:  PR[GP1:91,1] = PR[GP1:90,1] + -50.667;
   1:  PR[GP1:91,2] = PR[GP1:90,2] + -25.227;
   1:L PR[91] 10mm/sec CNT100;
   1:  PR[GP1:91,1] = PR[GP1:90,1] + -40.471;
   1:  PR[GP1:91,2] = PR[GP1:90,2] + -33.444;
   1:L PR[91] 10mm/sec CNT100;
   1:  PR[GP1:91,1] = PR[GP1:90,1] + -40.362;
   1:  PR[GP1:91,2] = PR[GP1:90,2] + -33.512;
   1:L PR[91] 10mm/sec CNT100;
   1:  PR[GP1:91,1] = PR[GP1:90,1] + -40.242;
   1:  PR[GP1:91,2] = PR[GP1:90,2] + -33.560;
   1:L PR[91] 10mm/sec CNT100;
   1:  PR[GP1:91,1] = PR[GP1:90,1] + -35.662;
   1:  PR[GP1:91,2] = PR[GP1:90,2] + -35.176;
   1:L PR[91] 10mm/sec CNT100;
   1:  PR[GP1:91,1] = PR[GP1:90,1] + -27.664;
   1:  PR[GP1:91,2] = PR[GP1:90,2] + -38.124;
   1:L PR[91] 10mm/sec CNT100;
   1:  PR[GP1:91,1] = PR[GP1:90,1] + -26.983;
   1:  PR[GP1:91,2] = PR[GP1:90,2] + -38.348;
   1:L PR[91] 10mm/sec CNT100;
   1:  PR[GP1:91,1] = PR[GP1:90,1] + -14.470;
   1:  PR[GP1:91,2] = PR[GP1:90,2] + -38.570;
   1:L PR[91] 10mm/sec CNT100;
   1:  PR[GP1:91,1] = PR[GP1:90,1] + -12.465;
   1:  PR[GP1:91,2] = PR[GP1:90,2] + -38.499;
   1:L PR[91] 10mm/sec CNT100;
   1:  PR[GP1:91,1] = PR[GP1:90,1] + -5.165;
   1:  PR[GP1:91,2] = PR[GP1:90,2] + -36.226;
   1:L PR[91] 10mm/sec CNT100;
   1:  PR[GP1:91,1] = PR[GP1:90,1] + -1.689;
   1:  PR[GP1:91,2] = PR[GP1:90,2] + -35.091;
   1:L PR[91] 10mm/sec CNT100;
   1:  PR[GP1:91,1] = PR[GP1:90,1] + 2.504;
   1:  PR[GP1:91,2] = PR[GP1:90,2] + -35.100;
   1:L PR[91] 10mm/sec CNT100;
   1:  PR[GP1:91,1] = PR[GP1:90,1] + 5.979;
   1:  PR[GP1:91,2] = PR[GP1:90,2] + -36.223;
   1:L PR[91] 10mm/sec CNT100;
   1:  PR[GP1:91,1] = PR[GP1:90,1] + 13.283;
   1:  PR[GP1:91,2] = PR[GP1:90,2] + -38.498;
   1:L PR[91] 10mm/sec CNT100;
   1:  PR[GP1:91,1] = PR[GP1:90,1] + 15.288;
   1:  PR[GP1:91,2] = PR[GP1:90,2] + -38.569;
   1:L PR[91] 10mm/sec CNT100;
   1:  PR[GP1:91,1] = PR[GP1:90,1] + 27.801;
   1:  PR[GP1:91,2] = PR[GP1:90,2] + -38.349;
   1:L PR[91] 10mm/sec CNT100;
   1:  PR[GP1:91,1] = PR[GP1:90,1] + 28.483;
   1:  PR[GP1:91,2] = PR[GP1:90,2] + -38.125;
   1:L PR[91] 10mm/sec CNT100;
   1:  PR[GP1:91,1] = PR[GP1:90,1] + 36.481;
   1:  PR[GP1:91,2] = PR[GP1:90,2] + -35.179;
   1:L PR[91] 10mm/sec CNT100;
   1:  PR[GP1:91,1] = PR[GP1:90,1] + 41.191;
   1:  PR[GP1:91,2] = PR[GP1:90,2] + -33.509;
   1:L PR[91] 10mm/sec CNT100;
   1:  PR[GP1:91,1] = PR[GP1:90,1] + 41.277;
   1:  PR[GP1:91,2] = PR[GP1:90,2] + -33.456;
   1:L PR[91] 10mm/sec CNT100;
   1:  PR[GP1:91,1] = PR[GP1:90,1] + 41.425;
   1:  PR[GP1:91,2] = PR[GP1:90,2] + -33.325;
   1:L PR[91] 10mm/sec CNT100;
   1:  PR[GP1:91,1] = PR[GP1:90,1] + 51.922;
   1:  PR[GP1:91,2] = PR[GP1:90,2] + -24.828;
   1:L PR[91] 10mm/sec CNT100;
   1:  PR[GP1:91,1] = PR[GP1:90,1] + 52.285;
   1:  PR[GP1:91,2] = PR[GP1:90,2] + -24.356;
   1:L PR[91] 10mm/sec CNT100;
   1:  PR[GP1:91,1] = PR[GP1:90,1] + 52.629;
   1:  PR[GP1:91,2] = PR[GP1:90,2] + -23.696;
   1:L PR[91] 10mm/sec CNT100;
   1:  PR[GP1:91,1] = PR[GP1:90,1] + 58.951;
   1:  PR[GP1:91,2] = PR[GP1:90,2] + -13.164;
   1:L PR[91] 10mm/sec CNT100;
   1:  PR[GP1:91,1] = PR[GP1:90,1] + 59.199;
   1:  PR[GP1:91,2] = PR[GP1:90,2] + -12.334;
   1:L PR[91] 10mm/sec CNT100;
   1:  PR[GP1:91,1] = PR[GP1:90,1] + 59.293;
   1:  PR[GP1:91,2] = PR[GP1:90,2] + -11.322;
   1:L PR[91] 10mm/sec CNT100;
   1:  PR[GP1:91,1] = PR[GP1:90,1] + 61.382;
   1:  PR[GP1:91,2] = PR[GP1:90,2] + 0.023;
   1:L PR[91] 10mm/sec CNT100;
   1:  PR[GP1:91,1] = PR[GP1:90,1] + 61.283;
   1:  PR[GP1:91,2] = PR[GP1:90,2] + 1.097;
   1:L PR[91] 10mm/sec CNT100;
   1:  PR[GP1:91,1] = PR[GP1:90,1] + 59.208;
   1:  PR[GP1:91,2] = PR[GP1:90,2] + 12.295;
   1:L PR[91] 10mm/sec CNT100;
   1:  PR[GP1:91,1] = PR[GP1:90,1] + 58.946;
   1:  PR[GP1:91,2] = PR[GP1:90,2] + 13.171;
   1:L PR[91] 10mm/sec CNT100;
   1:  PR[GP1:91,1] = PR[GP1:90,1] + 58.516;
   1:  PR[GP1:91,2] = PR[GP1:90,2] + 14.004;
   1:L PR[91] 10mm/sec CNT100;
   1:  PR[GP1:91,1] = PR[GP1:90,1] + 52.302;
   1:  PR[GP1:91,2] = PR[GP1:90,2] + 24.327;
   1:L PR[91] 10mm/sec CNT100;
   1:  PR[GP1:91,1] = PR[GP1:90,1] + 51.918;
   1:  PR[GP1:91,2] = PR[GP1:90,2] + 24.825;
   1:L PR[91] 10mm/sec CNT100;
   1:  PR[GP1:91,1] = PR[GP1:90,1] + 51.486;
   1:  PR[GP1:91,2] = PR[GP1:90,2] + 25.211;
   1:L PR[91] 10mm/sec CNT100;
   1:  PR[GP1:91,1] = PR[GP1:90,1] + 41.300;
   1:  PR[GP1:91,2] = PR[GP1:90,2] + 33.434;
   1:L PR[91] 10mm/sec CNT100;
   1:  PR[GP1:91,1] = PR[GP1:90,1] + 41.202;
   1:  PR[GP1:91,2] = PR[GP1:90,2] + 33.494;
   1:L PR[91] 10mm/sec CNT100;
   1:  PR[GP1:91,1] = PR[GP1:90,1] + 36.481;
   1:  PR[GP1:91,2] = PR[GP1:90,2] + 35.169;
   1:L PR[91] 10mm/sec CNT100;
   1:  PR[GP1:91,1] = PR[GP1:90,1] + 28.498;
   1:  PR[GP1:91,2] = PR[GP1:90,2] + 38.114;
   1:L PR[91] 10mm/sec CNT100;
   1:  PR[GP1:91,1] = PR[GP1:90,1] + 27.817;
   1:  PR[GP1:91,2] = PR[GP1:90,2] + 38.337;
   1:L PR[91] 10mm/sec CNT100;
   1:  PR[GP1:91,1] = PR[GP1:90,1] + 15.305;
   1:  PR[GP1:91,2] = PR[GP1:90,2] + 38.563;
   1:L PR[91] 10mm/sec CNT100;
   1:  PR[GP1:91,1] = PR[GP1:90,1] + 13.300;
   1:  PR[GP1:91,2] = PR[GP1:90,2] + 38.492;
   1:L PR[91] 10mm/sec CNT100;
   1:  PR[GP1:91,1] = PR[GP1:90,1] + 7.292;
   1:  PR[GP1:91,2] = PR[GP1:90,2] + 36.635;
   1:L PR[91] 10mm/sec CNT100;
   1:  PR[GP1:91,1] = PR[GP1:90,1] + 2.505;
   1:  PR[GP1:91,2] = PR[GP1:90,2] + 35.089;
   1:L PR[91] 10mm/sec CNT100;
   1:  PR[GP1:91,1] = PR[GP1:90,1] + -1.630;
   1:  PR[GP1:91,2] = PR[GP1:90,2] + 35.497;
   1:  PR[GP1:91,3] = PR[GP1:90,3] + 77.140;
   1:L PR[91] 10mm/sec CNT100;
   1:  PR[GP1:91,1] = PR[GP1:90,1] + -3.708;
   1:  PR[GP1:91,2] = PR[GP1:90,2] + 36.175;
   1:L PR[91] 10mm/sec CNT100;
   1:  PR[GP1:91,1] = PR[GP1:90,1] + -11.834;
   1:  PR[GP1:91,2] = PR[GP1:90,2] + 38.686;
   1:L PR[91] 10mm/sec CNT100;
   1:  PR[GP1:91,1] = PR[GP1:90,1] + -14.571;
   1:  PR[GP1:91,2] = PR[GP1:90,2] + 38.784;
   1:L PR[91] 10mm/sec CNT100;
   1:  PR[GP1:91,1] = PR[GP1:90,1] + -26.430;
   1:  PR[GP1:91,2] = PR[GP1:90,2] + 38.567;
   1:L PR[91] 10mm/sec CNT100;
   1:  PR[GP1:91,1] = PR[GP1:90,1] + -27.829;
   1:  PR[GP1:91,2] = PR[GP1:90,2] + 38.108;
   1:L PR[91] 10mm/sec CNT100;
   1:  PR[GP1:91,1] = PR[GP1:90,1] + -39.910;
   1:  PR[GP1:91,2] = PR[GP1:90,2] + 33.650;
   1:L PR[91] 10mm/sec CNT100;
   1:  PR[GP1:91,1] = PR[GP1:90,1] + -43.038;
   1:  PR[GP1:91,2] = PR[GP1:90,2] + 31.076;
   1:L PR[91] 10mm/sec CNT100;
   1:  PR[GP1:91,1] = PR[GP1:90,1] + -50.715;
   1:  PR[GP1:91,2] = PR[GP1:90,2] + 24.863;
   1:L PR[91] 10mm/sec CNT100;
   1:  PR[GP1:91,1] = PR[GP1:90,1] + -50.854;
   1:  PR[GP1:91,2] = PR[GP1:90,2] + 24.683;
   1:L PR[91] 10mm/sec CNT100;
   1:  PR[GP1:91,1] = PR[GP1:90,1] + -51.015;
   1:  PR[GP1:91,2] = PR[GP1:90,2] + 24.371;
   1:L PR[91] 10mm/sec CNT100;
   1:  PR[GP1:91,1] = PR[GP1:90,1] + -57.727;
   1:  PR[GP1:91,2] = PR[GP1:90,2] + 13.158;
   1:L PR[91] 10mm/sec CNT100;
   1:  PR[GP1:91,1] = PR[GP1:90,1] + -57.876;
   1:  PR[GP1:91,2] = PR[GP1:90,2] + 12.654;
   1:L PR[91] 10mm/sec CNT100;
   1:  PR[GP1:91,1] = PR[GP1:90,1] + -57.934;
   1:  PR[GP1:91,2] = PR[GP1:90,2] + 12.024;
   1:L PR[91] 10mm/sec CNT100;
   1:  PR[GP1:91,1] = PR[GP1:90,1] + -60.156;
   1:  PR[GP1:91,2] = PR[GP1:90,2] + -0.032;
   1:L PR[91] 10mm/sec CNT100;
   1:  PR[GP1:91,1] = PR[GP1:90,1] + -60.092;
   1:  PR[GP1:91,2] = PR[GP1:90,2] + -0.734;
   1:L PR[91] 10mm/sec CNT100;
   1:  PR[GP1:91,1] = PR[GP1:90,1] + -57.882;
   1:  PR[GP1:91,2] = PR[GP1:90,2] + -12.640;
   1:L PR[91] 10mm/sec CNT100;
   1:  PR[GP1:91,1] = PR[GP1:90,1] + -57.720;
   1:  PR[GP1:91,2] = PR[GP1:90,2] + -13.190;
   1:L PR[91] 10mm/sec CNT100;
   1:  PR[GP1:91,1] = PR[GP1:90,1] + -57.453;
   1:  PR[GP1:91,2] = PR[GP1:90,2] + -13.713;
   1:L PR[91] 10mm/sec CNT100;
   1:  PR[GP1:91,1] = PR[GP1:90,1] + -50.860;
   1:  PR[GP1:91,2] = PR[GP1:90,2] + -24.683;
   1:L PR[91] 10mm/sec CNT100;
   1:  PR[GP1:91,1] = PR[GP1:90,1] + -50.701;
   1:  PR[GP1:91,2] = PR[GP1:90,2] + -24.891;
   1:L PR[91] 10mm/sec CNT100;
   1:  PR[GP1:91,1] = PR[GP1:90,1] + -50.514;
   1:  PR[GP1:91,2] = PR[GP1:90,2] + -25.058;
   1:L PR[91] 10mm/sec CNT100;
   1:  PR[GP1:91,1] = PR[GP1:90,1] + -43.039;
   1:  PR[GP1:91,2] = PR[GP1:90,2] + -31.083;
   1:L PR[91] 10mm/sec CNT100;
   1:  PR[GP1:91,1] = PR[GP1:90,1] + -39.898;
   1:  PR[GP1:91,2] = PR[GP1:90,2] + -33.665;
   1:L PR[91] 10mm/sec CNT100;
   1:  PR[GP1:91,1] = PR[GP1:90,1] + -27.814;
   1:  PR[GP1:91,2] = PR[GP1:90,2] + -38.120;
   1:L PR[91] 10mm/sec CNT100;
   1:  PR[GP1:91,1] = PR[GP1:90,1] + -26.414;
   1:  PR[GP1:91,2] = PR[GP1:90,2] + -38.579;
   1:L PR[91] 10mm/sec CNT100;
   1:  PR[GP1:91,1] = PR[GP1:90,1] + -14.554;
   1:  PR[GP1:91,2] = PR[GP1:90,2] + -38.790;
   1:L PR[91] 10mm/sec CNT100;
   1:  PR[GP1:91,1] = PR[GP1:90,1] + -11.818;
   1:  PR[GP1:91,2] = PR[GP1:90,2] + -38.692;
   1:L PR[91] 10mm/sec CNT100;
   1:  PR[GP1:91,1] = PR[GP1:90,1] + -1.626;
   1:  PR[GP1:91,2] = PR[GP1:90,2] + -35.515;
   1:L PR[91] 10mm/sec CNT100;
   1:  PR[GP1:91,1] = PR[GP1:90,1] + 2.443;
   1:L PR[91] 10mm/sec CNT100;
   1:  PR[GP1:91,1] = PR[GP1:90,1] + 12.636;
   1:  PR[GP1:91,2] = PR[GP1:90,2] + -38.691;
   1:L PR[91] 10mm/sec CNT100;
   1:  PR[GP1:91,1] = PR[GP1:90,1] + 15.373;
   1:  PR[GP1:91,2] = PR[GP1:90,2] + -38.789;
   1:L PR[91] 10mm/sec CNT100;
   1:  PR[GP1:91,1] = PR[GP1:90,1] + 27.232;
   1:  PR[GP1:91,2] = PR[GP1:90,2] + -38.580;
   1:L PR[91] 10mm/sec CNT100;
   1:  PR[GP1:91,1] = PR[GP1:90,1] + 28.633;
   1:  PR[GP1:91,2] = PR[GP1:90,2] + -38.120;
   1:L PR[91] 10mm/sec CNT100;
   1:  PR[GP1:91,1] = PR[GP1:90,1] + 40.717;
   1:  PR[GP1:91,2] = PR[GP1:90,2] + -33.669;
   1:L PR[91] 10mm/sec CNT100;
   1:  PR[GP1:91,1] = PR[GP1:90,1] + 43.858;
   1:  PR[GP1:91,2] = PR[GP1:90,2] + -31.083;
   1:L PR[91] 10mm/sec CNT100;
   1:  PR[GP1:91,1] = PR[GP1:90,1] + 51.526;
   1:  PR[GP1:91,2] = PR[GP1:90,2] + -24.877;
   1:L PR[91] 10mm/sec CNT100;
   1:  PR[GP1:91,1] = PR[GP1:90,1] + 51.667;
   1:  PR[GP1:91,2] = PR[GP1:90,2] + -24.694;
   1:L PR[91] 10mm/sec CNT100;
   1:  PR[GP1:91,1] = PR[GP1:90,1] + 51.828;
   1:  PR[GP1:91,2] = PR[GP1:90,2] + -24.384;
   1:L PR[91] 10mm/sec CNT100;
   1:  PR[GP1:91,1] = PR[GP1:90,1] + 58.544;
   1:  PR[GP1:91,2] = PR[GP1:90,2] + -13.195;
   1:L PR[91] 10mm/sec CNT100;
   1:  PR[GP1:91,1] = PR[GP1:90,1] + 58.692;
   1:  PR[GP1:91,2] = PR[GP1:90,2] + -12.699;
   1:L PR[91] 10mm/sec CNT100;
   1:  PR[GP1:91,1] = PR[GP1:90,1] + 58.753;
   1:  PR[GP1:91,2] = PR[GP1:90,2] + -12.052;
   1:L PR[91] 10mm/sec CNT100;
   1:  PR[GP1:91,1] = PR[GP1:90,1] + 60.976;
   1:  PR[GP1:91,2] = PR[GP1:90,2] + 0.023;
   1:L PR[91] 10mm/sec CNT100;
   1:  PR[GP1:91,1] = PR[GP1:90,1] + 60.910;
   1:  PR[GP1:91,2] = PR[GP1:90,2] + 0.747;
   1:L PR[91] 10mm/sec CNT100;
   1:  PR[GP1:91,1] = PR[GP1:90,1] + 58.701;
   1:  PR[GP1:91,2] = PR[GP1:90,2] + 12.661;
   1:L PR[91] 10mm/sec CNT100;
   1:  PR[GP1:91,1] = PR[GP1:90,1] + 58.540;
   1:  PR[GP1:91,2] = PR[GP1:90,2] + 13.201;
   1:L PR[91] 10mm/sec CNT100;
   1:  PR[GP1:91,1] = PR[GP1:90,1] + 58.272;
   1:  PR[GP1:91,2] = PR[GP1:90,2] + 13.720;
   1:L PR[91] 10mm/sec CNT100;
   1:  PR[GP1:91,1] = PR[GP1:90,1] + 51.683;
   1:  PR[GP1:91,2] = PR[GP1:90,2] + 24.664;
   1:L PR[91] 10mm/sec CNT100;
   1:  PR[GP1:91,1] = PR[GP1:90,1] + 51.522;
   1:  PR[GP1:91,2] = PR[GP1:90,2] + 24.873;
   1:L PR[91] 10mm/sec CNT100;
   1:  PR[GP1:91,1] = PR[GP1:90,1] + 51.336;
   1:  PR[GP1:91,2] = PR[GP1:90,2] + 25.040;
   1:L PR[91] 10mm/sec CNT100;
   1:  PR[GP1:91,1] = PR[GP1:90,1] + 43.858;
   1:  PR[GP1:91,2] = PR[GP1:90,2] + 31.076;
   1:L PR[91] 10mm/sec CNT100;
   1:  PR[GP1:91,1] = PR[GP1:90,1] + 40.728;
   1:  PR[GP1:91,2] = PR[GP1:90,2] + 33.654;
   1:L PR[91] 10mm/sec CNT100;
   1:  PR[GP1:91,1] = PR[GP1:90,1] + 28.647;
   1:  PR[GP1:91,2] = PR[GP1:90,2] + 38.109;
   1:L PR[91] 10mm/sec CNT100;
   1:  PR[GP1:91,1] = PR[GP1:90,1] + 27.248;
   1:  PR[GP1:91,2] = PR[GP1:90,2] + 38.568;
   1:L PR[91] 10mm/sec CNT100;
   1:  PR[GP1:91,1] = PR[GP1:90,1] + 15.389;
   1:  PR[GP1:91,2] = PR[GP1:90,2] + 38.783;
   1:L PR[91] 10mm/sec CNT100;
   1:  PR[GP1:91,1] = PR[GP1:90,1] + 12.651;
   1:  PR[GP1:91,2] = PR[GP1:90,2] + 38.685;
   1:L PR[91] 10mm/sec CNT100;
   1:  PR[GP1:91,1] = PR[GP1:90,1] + 4.522;
   1:  PR[GP1:91,2] = PR[GP1:90,2] + 36.172;
   1:L PR[91] 10mm/sec CNT100;
   1:  PR[GP1:91,1] = PR[GP1:90,1] + 2.447;
   1:  PR[GP1:91,2] = PR[GP1:90,2] + 35.502;
   1:L PR[91] 10mm/sec CNT100;
   1:  PR[GP1:91,1] = PR[GP1:90,1] + -1.568;
   1:  PR[GP1:91,2] = PR[GP1:90,2] + 35.907;
   1:  PR[GP1:91,3] = PR[GP1:90,3] + 78.470;
   1:L PR[91] 10mm/sec CNT100;
   1:  PR[GP1:91,1] = PR[GP1:90,1] + -11.185;
   1:  PR[GP1:91,2] = PR[GP1:90,2] + 38.879;
   1:L PR[91] 10mm/sec CNT100;
   1:  PR[GP1:91,1] = PR[GP1:90,1] + -14.654;
   1:  PR[GP1:91,2] = PR[GP1:90,2] + 39.003;
   1:L PR[91] 10mm/sec CNT100;
   1:  PR[GP1:91,1] = PR[GP1:90,1] + -25.860;
   1:  PR[GP1:91,2] = PR[GP1:90,2] + 38.799;
   1:L PR[91] 10mm/sec CNT100;
   1:  PR[GP1:91,1] = PR[GP1:90,1] + -27.978;
   1:  PR[GP1:91,2] = PR[GP1:90,2] + 38.104;
   1:L PR[91] 10mm/sec CNT100;
   1:  PR[GP1:91,1] = PR[GP1:90,1] + -39.432;
   1:  PR[GP1:91,2] = PR[GP1:90,2] + 33.877;
   1:L PR[91] 10mm/sec CNT100;
   1:  PR[GP1:91,1] = PR[GP1:90,1] + -40.210;
   1:  PR[GP1:91,2] = PR[GP1:90,2] + 33.261;
   1:L PR[91] 10mm/sec CNT100;
   1:  PR[GP1:91,1] = PR[GP1:90,1] + -50.286;
   1:  PR[GP1:91,2] = PR[GP1:90,2] + 24.945;
   1:L PR[91] 10mm/sec CNT100;
   1:  PR[GP1:91,1] = PR[GP1:90,1] + -57.319;
   1:  PR[GP1:91,2] = PR[GP1:90,2] + 13.192;
   1:L PR[91] 10mm/sec CNT100;
   1:  PR[GP1:91,1] = PR[GP1:90,1] + -57.368;
   1:  PR[GP1:91,2] = PR[GP1:90,2] + 13.028;
   1:L PR[91] 10mm/sec CNT100;
   1:  PR[GP1:91,1] = PR[GP1:90,1] + -57.393;
   1:  PR[GP1:91,2] = PR[GP1:90,2] + 12.753;
   1:L PR[91] 10mm/sec CNT100;
   1:  PR[GP1:91,1] = PR[GP1:90,1] + -59.750;
   1:  PR[GP1:91,2] = PR[GP1:90,2] + -0.032;
   1:L PR[91] 10mm/sec CNT100;
   1:  PR[GP1:91,1] = PR[GP1:90,1] + -59.717;
   1:  PR[GP1:91,2] = PR[GP1:90,2] + -0.393;
   1:L PR[91] 10mm/sec CNT100;
   1:  PR[GP1:91,1] = PR[GP1:90,1] + -57.374;
   1:  PR[GP1:91,2] = PR[GP1:90,2] + -13.014;
   1:L PR[91] 10mm/sec CNT100;
   1:  PR[GP1:91,1] = PR[GP1:90,1] + -57.312;
   1:  PR[GP1:91,2] = PR[GP1:90,2] + -13.225;
   1:L PR[91] 10mm/sec CNT100;
   1:  PR[GP1:91,1] = PR[GP1:90,1] + -57.207;
   1:  PR[GP1:91,2] = PR[GP1:90,2] + -13.431;
   1:L PR[91] 10mm/sec CNT100;
   1:  PR[GP1:91,1] = PR[GP1:90,1] + -50.281;
   1:  PR[GP1:91,2] = PR[GP1:90,2] + -24.960;
   1:L PR[91] 10mm/sec CNT100;
   1:  PR[GP1:91,1] = PR[GP1:90,1] + -40.200;
   1:  PR[GP1:91,2] = PR[GP1:90,2] + -33.276;
   1:L PR[91] 10mm/sec CNT100;
   1:  PR[GP1:91,1] = PR[GP1:90,1] + -39.421;
   1:  PR[GP1:91,2] = PR[GP1:90,2] + -33.892;
   1:L PR[91] 10mm/sec CNT100;
   1:  PR[GP1:91,1] = PR[GP1:90,1] + -27.964;
   1:  PR[GP1:91,2] = PR[GP1:90,2] + -38.115;
   1:L PR[91] 10mm/sec CNT100;
   1:  PR[GP1:91,1] = PR[GP1:90,1] + -25.845;
   1:  PR[GP1:91,2] = PR[GP1:90,2] + -38.810;
   1:L PR[91] 10mm/sec CNT100;
   1:  PR[GP1:91,1] = PR[GP1:90,1] + -14.639;
   1:  PR[GP1:91,2] = PR[GP1:90,2] + -39.009;
   1:L PR[91] 10mm/sec CNT100;
   1:  PR[GP1:91,1] = PR[GP1:90,1] + -11.170;
   1:  PR[GP1:91,2] = PR[GP1:90,2] + -38.886;
   1:L PR[91] 10mm/sec CNT100;
   1:  PR[GP1:91,1] = PR[GP1:90,1] + -1.571;
   1:  PR[GP1:91,2] = PR[GP1:90,2] + -35.897;
   1:L PR[91] 10mm/sec CNT100;
   1:  PR[GP1:91,1] = PR[GP1:90,1] + 2.388;
   1:  PR[GP1:91,2] = PR[GP1:90,2] + -35.896;
   1:L PR[91] 10mm/sec CNT100;
   1:  PR[GP1:91,1] = PR[GP1:90,1] + 11.989;
   1:  PR[GP1:91,2] = PR[GP1:90,2] + -38.885;
   1:L PR[91] 10mm/sec CNT100;
   1:  PR[GP1:91,1] = PR[GP1:90,1] + 15.457;
   1:  PR[GP1:91,2] = PR[GP1:90,2] + -39.009;
   1:L PR[91] 10mm/sec CNT100;
   1:  PR[GP1:91,1] = PR[GP1:90,1] + 26.664;
   1:  PR[GP1:91,2] = PR[GP1:90,2] + -38.811;
   1:L PR[91] 10mm/sec CNT100;
   1:  PR[GP1:91,1] = PR[GP1:90,1] + 28.783;
   1:  PR[GP1:91,2] = PR[GP1:90,2] + -38.116;
   1:L PR[91] 10mm/sec CNT100;
   1:  PR[GP1:91,1] = PR[GP1:90,1] + 40.241;
   1:  PR[GP1:91,2] = PR[GP1:90,2] + -33.895;
   1:L PR[91] 10mm/sec CNT100;
   1:  PR[GP1:91,1] = PR[GP1:90,1] + 41.020;
   1:  PR[GP1:91,2] = PR[GP1:90,2] + -33.279;
   1:L PR[91] 10mm/sec CNT100;
   1:  PR[GP1:91,1] = PR[GP1:90,1] + 51.101;
   1:  PR[GP1:91,2] = PR[GP1:90,2] + -24.954;
   1:L PR[91] 10mm/sec CNT100;
   1:  PR[GP1:91,1] = PR[GP1:90,1] + 58.138;
   1:  PR[GP1:91,2] = PR[GP1:90,2] + -13.225;
   1:L PR[91] 10mm/sec CNT100;
   1:  PR[GP1:91,1] = PR[GP1:90,1] + 58.186;
   1:  PR[GP1:91,2] = PR[GP1:90,2] + -13.065;
   1:L PR[91] 10mm/sec CNT100;
   1:  PR[GP1:91,1] = PR[GP1:90,1] + 58.212;
   1:  PR[GP1:91,2] = PR[GP1:90,2] + -12.782;
   1:L PR[91] 10mm/sec CNT100;
   1:  PR[GP1:91,1] = PR[GP1:90,1] + 60.570;
   1:  PR[GP1:91,2] = PR[GP1:90,2] + 0.023;
   1:L PR[91] 10mm/sec CNT100;
   1:  PR[GP1:91,1] = PR[GP1:90,1] + 60.536;
   1:  PR[GP1:91,2] = PR[GP1:90,2] + 0.396;
   1:L PR[91] 10mm/sec CNT100;
   1:  PR[GP1:91,1] = PR[GP1:90,1] + 58.195;
   1:  PR[GP1:91,2] = PR[GP1:90,2] + 13.026;
   1:L PR[91] 10mm/sec CNT100;
   1:  PR[GP1:91,1] = PR[GP1:90,1] + 58.134;
   1:  PR[GP1:91,2] = PR[GP1:90,2] + 13.231;
   1:L PR[91] 10mm/sec CNT100;
   1:  PR[GP1:91,1] = PR[GP1:90,1] + 58.028;
   1:  PR[GP1:91,2] = PR[GP1:90,2] + 13.436;
   1:L PR[91] 10mm/sec CNT100;
   1:  PR[GP1:91,1] = PR[GP1:90,1] + 51.106;
   1:  PR[GP1:91,2] = PR[GP1:90,2] + 24.938;
   1:L PR[91] 10mm/sec CNT100;
   1:  PR[GP1:91,1] = PR[GP1:90,1] + 41.029;
   1:  PR[GP1:91,2] = PR[GP1:90,2] + 33.264;
   1:L PR[91] 10mm/sec CNT100;
   1:  PR[GP1:91,1] = PR[GP1:90,1] + 40.251;
   1:  PR[GP1:91,2] = PR[GP1:90,2] + 33.880;
   1:L PR[91] 10mm/sec CNT100;
   1:  PR[GP1:91,1] = PR[GP1:90,1] + 28.796;
   1:  PR[GP1:91,2] = PR[GP1:90,2] + 38.105;
   1:L PR[91] 10mm/sec CNT100;
   1:  PR[GP1:91,1] = PR[GP1:90,1] + 26.678;
   1:  PR[GP1:91,2] = PR[GP1:90,2] + 38.800;
   1:L PR[91] 10mm/sec CNT100;
   1:  PR[GP1:91,1] = PR[GP1:90,1] + 15.472;
   1:  PR[GP1:91,2] = PR[GP1:90,2] + 39.002;
   1:L PR[91] 10mm/sec CNT100;
   1:  PR[GP1:91,1] = PR[GP1:90,1] + 12.003;
   1:  PR[GP1:91,2] = PR[GP1:90,2] + 38.878;
   1:L PR[91] 10mm/sec CNT100;
   1:  PR[GP1:91,1] = PR[GP1:90,1] + 2.386;
   1:  PR[GP1:91,2] = PR[GP1:90,2] + 35.906;
   1:L PR[91] 10mm/sec CNT100;
   1:  PR[GP1:91,1] = PR[GP1:90,1] + -1.513;
   1:  PR[GP1:91,2] = PR[GP1:90,2] + 36.285;
   1:  PR[GP1:91,3] = PR[GP1:90,3] + 79.800;
   1:L PR[91] 10mm/sec CNT100;
   1:  PR[GP1:91,1] = PR[GP1:90,1] + -10.536;
   1:  PR[GP1:91,2] = PR[GP1:90,2] + 39.072;
   1:L PR[91] 10mm/sec CNT100;
   1:  PR[GP1:91,1] = PR[GP1:90,1] + -14.737;
   1:  PR[GP1:91,2] = PR[GP1:90,2] + 39.223;
   1:L PR[91] 10mm/sec CNT100;
   1:  PR[GP1:91,1] = PR[GP1:90,1] + -25.290;
   1:  PR[GP1:91,2] = PR[GP1:90,2] + 39.030;
   1:L PR[91] 10mm/sec CNT100;
   1:  PR[GP1:91,1] = PR[GP1:90,1] + -28.127;
   1:  PR[GP1:91,2] = PR[GP1:90,2] + 38.100;
   1:L PR[91] 10mm/sec CNT100;
   1:  PR[GP1:91,1] = PR[GP1:90,1] + -38.949;
   1:  PR[GP1:91,2] = PR[GP1:90,2] + 34.106;
   1:L PR[91] 10mm/sec CNT100;
   1:  PR[GP1:91,1] = PR[GP1:90,1] + -40.341;
   1:  PR[GP1:91,2] = PR[GP1:90,2] + 33.005;
   1:L PR[91] 10mm/sec CNT100;
   1:  PR[GP1:91,1] = PR[GP1:90,1] + -49.882;
   1:  PR[GP1:91,2] = PR[GP1:90,2] + 25.129;
   1:L PR[91] 10mm/sec CNT100;
   1:  PR[GP1:91,1] = PR[GP1:90,1] + -56.903;
   1:  PR[GP1:91,2] = PR[GP1:90,2] + 13.265;
   1:L PR[91] 10mm/sec CNT100;
   1:  PR[GP1:91,1] = PR[GP1:90,1] + -57.532;
   1:  PR[GP1:91,2] = PR[GP1:90,2] + 9.793;
   1:L PR[91] 10mm/sec CNT100;
   1:  PR[GP1:91,1] = PR[GP1:90,1] + -59.343;
   1:  PR[GP1:91,2] = PR[GP1:90,2] + -0.032;
   1:L PR[91] 10mm/sec CNT100;
   1:  PR[GP1:91,1] = PR[GP1:90,1] + -59.342;
   1:  PR[GP1:91,2] = PR[GP1:90,2] + -0.052;
   1:L PR[91] 10mm/sec CNT100;
   1:  PR[GP1:91,1] = PR[GP1:90,1] + -57.532;
   1:  PR[GP1:91,2] = PR[GP1:90,2] + -9.801;
   1:L PR[91] 10mm/sec CNT100;
   1:  PR[GP1:91,1] = PR[GP1:90,1] + -56.901;
   1:  PR[GP1:91,2] = PR[GP1:90,2] + -13.278;
   1:L PR[91] 10mm/sec CNT100;
   1:  PR[GP1:91,1] = PR[GP1:90,1] + -49.877;
   1:  PR[GP1:91,2] = PR[GP1:90,2] + -25.144;
   1:L PR[91] 10mm/sec CNT100;
   1:  PR[GP1:91,1] = PR[GP1:90,1] + -40.331;
   1:  PR[GP1:91,2] = PR[GP1:90,2] + -33.019;
   1:L PR[91] 10mm/sec CNT100;
   1:  PR[GP1:91,1] = PR[GP1:90,1] + -38.939;
   1:  PR[GP1:91,2] = PR[GP1:90,2] + -34.120;
   1:L PR[91] 10mm/sec CNT100;
   1:  PR[GP1:91,1] = PR[GP1:90,1] + -28.115;
   1:  PR[GP1:91,2] = PR[GP1:90,2] + -38.111;
   1:L PR[91] 10mm/sec CNT100;
   1:  PR[GP1:91,1] = PR[GP1:90,1] + -25.276;
   1:  PR[GP1:91,2] = PR[GP1:90,2] + -39.042;
   1:L PR[91] 10mm/sec CNT100;
   1:  PR[GP1:91,1] = PR[GP1:90,1] + -14.723;
   1:  PR[GP1:91,2] = PR[GP1:90,2] + -39.229;
   1:L PR[91] 10mm/sec CNT100;
   1:  PR[GP1:91,1] = PR[GP1:90,1] + -10.523;
   1:  PR[GP1:91,2] = PR[GP1:90,2] + -39.079;
   1:L PR[91] 10mm/sec CNT100;
   1:  PR[GP1:91,1] = PR[GP1:90,1] + -1.515;
   1:  PR[GP1:91,2] = PR[GP1:90,2] + -36.276;
   1:L PR[91] 10mm/sec CNT100;
   1:  PR[GP1:91,1] = PR[GP1:90,1] + 2.333;
   1:  PR[GP1:91,2] = PR[GP1:90,2] + -36.275;
   1:L PR[91] 10mm/sec CNT100;
   1:  PR[GP1:91,1] = PR[GP1:90,1] + 11.342;
   1:  PR[GP1:91,2] = PR[GP1:90,2] + -39.079;
   1:L PR[91] 10mm/sec CNT100;
   1:  PR[GP1:91,1] = PR[GP1:90,1] + 15.542;
   1:  PR[GP1:91,2] = PR[GP1:90,2] + -39.228;
   1:L PR[91] 10mm/sec CNT100;
   1:  PR[GP1:91,1] = PR[GP1:90,1] + 26.095;
   1:  PR[GP1:91,2] = PR[GP1:90,2] + -39.042;
   1:L PR[91] 10mm/sec CNT100;
   1:  PR[GP1:91,1] = PR[GP1:90,1] + 28.933;
   1:  PR[GP1:91,2] = PR[GP1:90,2] + -38.111;
   1:L PR[91] 10mm/sec CNT100;
   1:  PR[GP1:91,1] = PR[GP1:90,1] + 39.758;
   1:  PR[GP1:91,2] = PR[GP1:90,2] + -34.123;
   1:L PR[91] 10mm/sec CNT100;
   1:  PR[GP1:91,1] = PR[GP1:90,1] + 41.150;
   1:  PR[GP1:91,2] = PR[GP1:90,2] + -33.021;
   1:L PR[91] 10mm/sec CNT100;
   1:  PR[GP1:91,1] = PR[GP1:90,1] + 50.699;
   1:  PR[GP1:91,2] = PR[GP1:90,2] + -25.137;
   1:L PR[91] 10mm/sec CNT100;
   1:  PR[GP1:91,1] = PR[GP1:90,1] + 51.075;
   1:  PR[GP1:91,2] = PR[GP1:90,2] + -24.515;
   1:L PR[91] 10mm/sec CNT100;
   1:  PR[GP1:91,1] = PR[GP1:90,1] + 57.722;
   1:  PR[GP1:91,2] = PR[GP1:90,2] + -13.296;
   1:L PR[91] 10mm/sec CNT100;
   1:  PR[GP1:91,1] = PR[GP1:90,1] + 60.164;
   1:  PR[GP1:91,2] = PR[GP1:90,2] + 0.023;
   1:L PR[91] 10mm/sec CNT100;
   1:  PR[GP1:91,1] = PR[GP1:90,1] + 60.162;
   1:  PR[GP1:91,2] = PR[GP1:90,2] + 0.046;
   1:L PR[91] 10mm/sec CNT100;
   1:  PR[GP1:91,1] = PR[GP1:90,1] + 58.352;
   1:  PR[GP1:91,2] = PR[GP1:90,2] + 9.809;
   1:L PR[91] 10mm/sec CNT100;
   1:  PR[GP1:91,1] = PR[GP1:90,1] + 57.723;
   1:  PR[GP1:91,2] = PR[GP1:90,2] + 13.283;
   1:L PR[91] 10mm/sec CNT100;
   1:  PR[GP1:91,1] = PR[GP1:90,1] + 50.702;
   1:  PR[GP1:91,2] = PR[GP1:90,2] + 25.123;
   1:L PR[91] 10mm/sec CNT100;
   1:  PR[GP1:91,1] = PR[GP1:90,1] + 41.160;
   1:  PR[GP1:91,2] = PR[GP1:90,2] + 33.008;
   1:L PR[91] 10mm/sec CNT100;
   1:  PR[GP1:91,1] = PR[GP1:90,1] + 39.768;
   1:  PR[GP1:91,2] = PR[GP1:90,2] + 34.109;
   1:L PR[91] 10mm/sec CNT100;
   1:  PR[GP1:91,1] = PR[GP1:90,1] + 28.946;
   1:  PR[GP1:91,2] = PR[GP1:90,2] + 38.100;
   1:L PR[91] 10mm/sec CNT100;
   1:  PR[GP1:91,1] = PR[GP1:90,1] + 26.108;
   1:  PR[GP1:91,2] = PR[GP1:90,2] + 39.031;
   1:L PR[91] 10mm/sec CNT100;
   1:  PR[GP1:91,1] = PR[GP1:90,1] + 15.556;
   1:  PR[GP1:91,2] = PR[GP1:90,2] + 39.222;
   1:L PR[91] 10mm/sec CNT100;
   1:  PR[GP1:91,1] = PR[GP1:90,1] + 11.354;
   1:  PR[GP1:91,2] = PR[GP1:90,2] + 39.071;
   1:L PR[91] 10mm/sec CNT100;
   1:  PR[GP1:91,1] = PR[GP1:90,1] + 2.331;
   1:  PR[GP1:91,2] = PR[GP1:90,2] + 36.284;
   1:L PR[91] 10mm/sec CNT100;
   1:  PR[GP1:91,1] = PR[GP1:90,1] + -1.458;
   1:  PR[GP1:91,2] = PR[GP1:90,2] + 36.663;
   1:  PR[GP1:91,3] = PR[GP1:90,3] + 81.130;
   1:L PR[91] 10mm/sec CNT100;
   1:  PR[GP1:91,1] = PR[GP1:90,1] + -9.887;
   1:  PR[GP1:91,2] = PR[GP1:90,2] + 39.265;
   1:L PR[91] 10mm/sec CNT100;
   1:  PR[GP1:91,1] = PR[GP1:90,1] + -14.821;
   1:  PR[GP1:91,2] = PR[GP1:90,2] + 39.442;
   1:L PR[91] 10mm/sec CNT100;
   1:  PR[GP1:91,1] = PR[GP1:90,1] + -24.720;
   1:  PR[GP1:91,2] = PR[GP1:90,2] + 39.262;
   1:L PR[91] 10mm/sec CNT100;
   1:  PR[GP1:91,1] = PR[GP1:90,1] + -28.277;
   1:  PR[GP1:91,2] = PR[GP1:90,2] + 38.095;
   1:L PR[91] 10mm/sec CNT100;
   1:  PR[GP1:91,1] = PR[GP1:90,1] + -38.466;
   1:  PR[GP1:91,2] = PR[GP1:90,2] + 34.335;
   1:L PR[91] 10mm/sec CNT100;
   1:  PR[GP1:91,1] = PR[GP1:90,1] + -40.471;
   1:  PR[GP1:91,2] = PR[GP1:90,2] + 32.748;
   1:L PR[91] 10mm/sec CNT100;
   1:  PR[GP1:91,1] = PR[GP1:90,1] + -49.482;
   1:  PR[GP1:91,2] = PR[GP1:90,2] + 25.311;
   1:L PR[91] 10mm/sec CNT100;
   1:  PR[GP1:91,1] = PR[GP1:90,1] + -50.275;
   1:  PR[GP1:91,2] = PR[GP1:90,2] + 23.999;
   1:L PR[91] 10mm/sec CNT100;
   1:  PR[GP1:91,1] = PR[GP1:90,1] + -56.557;
   1:  PR[GP1:91,2] = PR[GP1:90,2] + 13.369;
   1:L PR[91] 10mm/sec CNT100;
   1:  PR[GP1:91,1] = PR[GP1:90,1] + -58.905;
   1:  PR[GP1:91,2] = PR[GP1:90,2] + 0.420;
   1:L PR[91] 10mm/sec CNT100;
   1:  PR[GP1:91,1] = PR[GP1:90,1] + -58.972;
   1:  PR[GP1:91,2] = PR[GP1:90,2] + 0.002;
   1:L PR[91] 10mm/sec CNT100;
   1:  PR[GP1:91,1] = PR[GP1:90,1] + -56.806;
   1:  PR[GP1:91,2] = PR[GP1:90,2] + -11.897;
   1:L PR[91] 10mm/sec CNT100;
   1:  PR[GP1:91,1] = PR[GP1:90,1] + -56.705;
   1:  PR[GP1:91,2] = PR[GP1:90,2] + -12.572;
   1:L PR[91] 10mm/sec CNT100;
   1:  PR[GP1:91,1] = PR[GP1:90,1] + -56.556;
   1:  PR[GP1:91,2] = PR[GP1:90,2] + -13.380;
   1:L PR[91] 10mm/sec CNT100;
   1:  PR[GP1:91,1] = PR[GP1:90,1] + -50.270;
   1:  PR[GP1:91,2] = PR[GP1:90,2] + -24.013;
   1:L PR[91] 10mm/sec CNT100;
   1:  PR[GP1:91,1] = PR[GP1:90,1] + -49.477;
   1:  PR[GP1:91,2] = PR[GP1:90,2] + -25.326;
   1:L PR[91] 10mm/sec CNT100;
   1:  PR[GP1:91,1] = PR[GP1:90,1] + -40.463;
   1:  PR[GP1:91,2] = PR[GP1:90,2] + -32.762;
   1:L PR[91] 10mm/sec CNT100;
   1:  PR[GP1:91,1] = PR[GP1:90,1] + -38.457;
   1:  PR[GP1:91,2] = PR[GP1:90,2] + -34.349;
   1:L PR[91] 10mm/sec CNT100;
   1:  PR[GP1:91,1] = PR[GP1:90,1] + -28.265;
   1:  PR[GP1:91,2] = PR[GP1:90,2] + -38.106;
   1:L PR[91] 10mm/sec CNT100;
   1:  PR[GP1:91,1] = PR[GP1:90,1] + -24.708;
   1:  PR[GP1:91,2] = PR[GP1:90,2] + -39.273;
   1:L PR[91] 10mm/sec CNT100;
   1:  PR[GP1:91,1] = PR[GP1:90,1] + -14.807;
   1:  PR[GP1:91,2] = PR[GP1:90,2] + -39.449;
   1:L PR[91] 10mm/sec CNT100;
   1:  PR[GP1:91,1] = PR[GP1:90,1] + -9.875;
   1:  PR[GP1:91,2] = PR[GP1:90,2] + -39.273;
   1:L PR[91] 10mm/sec CNT100;
   1:  PR[GP1:91,1] = PR[GP1:90,1] + -1.460;
   1:  PR[GP1:91,2] = PR[GP1:90,2] + -36.655;
   1:L PR[91] 10mm/sec CNT100;
   1:  PR[GP1:91,1] = PR[GP1:90,1] + 2.279;
   1:  PR[GP1:91,2] = PR[GP1:90,2] + -36.654;
   1:L PR[91] 10mm/sec CNT100;
   1:  PR[GP1:91,1] = PR[GP1:90,1] + 10.695;
   1:  PR[GP1:91,2] = PR[GP1:90,2] + -39.272;
   1:L PR[91] 10mm/sec CNT100;
   1:  PR[GP1:91,1] = PR[GP1:90,1] + 15.627;
   1:  PR[GP1:91,2] = PR[GP1:90,2] + -39.448;
   1:L PR[91] 10mm/sec CNT100;
   1:  PR[GP1:91,1] = PR[GP1:90,1] + 25.527;
   1:  PR[GP1:91,2] = PR[GP1:90,2] + -39.273;
   1:L PR[91] 10mm/sec CNT100;
   1:  PR[GP1:91,1] = PR[GP1:90,1] + 29.084;
   1:  PR[GP1:91,2] = PR[GP1:90,2] + -38.106;
   1:L PR[91] 10mm/sec CNT100;
   1:  PR[GP1:91,1] = PR[GP1:90,1] + 39.276;
   1:  PR[GP1:91,2] = PR[GP1:90,2] + -34.352;
   1:L PR[91] 10mm/sec CNT100;
   1:  PR[GP1:91,1] = PR[GP1:90,1] + 41.282;
   1:  PR[GP1:91,2] = PR[GP1:90,2] + -32.764;
   1:L PR[91] 10mm/sec CNT100;
   1:  PR[GP1:91,1] = PR[GP1:90,1] + 50.297;
   1:  PR[GP1:91,2] = PR[GP1:90,2] + -25.320;
   1:L PR[91] 10mm/sec CNT100;
   1:  PR[GP1:91,1] = PR[GP1:90,1] + 51.091;
   1:  PR[GP1:91,2] = PR[GP1:90,2] + -24.007;
   1:L PR[91] 10mm/sec CNT100;
   1:  PR[GP1:91,1] = PR[GP1:90,1] + 57.376;
   1:  PR[GP1:91,2] = PR[GP1:90,2] + -13.398;
   1:L PR[91] 10mm/sec CNT100;
   1:  PR[GP1:91,1] = PR[GP1:90,1] + 59.792;
   1:  PR[GP1:91,2] = PR[GP1:90,2] + -0.005;
   1:L PR[91] 10mm/sec CNT100;
   1:  PR[GP1:91,1] = PR[GP1:90,1] + 57.628;
   1:  PR[GP1:91,2] = PR[GP1:90,2] + 11.901;
   1:L PR[91] 10mm/sec CNT100;
   1:  PR[GP1:91,1] = PR[GP1:90,1] + 57.527;
   1:  PR[GP1:91,2] = PR[GP1:90,2] + 12.576;
   1:L PR[91] 10mm/sec CNT100;
   1:  PR[GP1:91,1] = PR[GP1:90,1] + 57.378;
   1:  PR[GP1:91,2] = PR[GP1:90,2] + 13.385;
   1:L PR[91] 10mm/sec CNT100;
   1:  PR[GP1:91,1] = PR[GP1:90,1] + 51.096;
   1:  PR[GP1:91,2] = PR[GP1:90,2] + 23.993;
   1:L PR[91] 10mm/sec CNT100;
   1:  PR[GP1:91,1] = PR[GP1:90,1] + 50.302;
   1:  PR[GP1:91,2] = PR[GP1:90,2] + 25.305;
   1:L PR[91] 10mm/sec CNT100;
   1:  PR[GP1:91,1] = PR[GP1:90,1] + 41.291;
   1:  PR[GP1:91,2] = PR[GP1:90,2] + 32.751;
   1:L PR[91] 10mm/sec CNT100;
   1:  PR[GP1:91,1] = PR[GP1:90,1] + 39.285;
   1:  PR[GP1:91,2] = PR[GP1:90,2] + 34.338;
   1:L PR[91] 10mm/sec CNT100;
   1:  PR[GP1:91,1] = PR[GP1:90,1] + 29.095;
   1:  PR[GP1:91,2] = PR[GP1:90,2] + 38.096;
   1:L PR[91] 10mm/sec CNT100;
   1:  PR[GP1:91,1] = PR[GP1:90,1] + 25.539;
   1:  PR[GP1:91,2] = PR[GP1:90,2] + 39.262;
   1:L PR[91] 10mm/sec CNT100;
   1:  PR[GP1:91,1] = PR[GP1:90,1] + 15.639;
   1:  PR[GP1:91,2] = PR[GP1:90,2] + 39.442;
   1:L PR[91] 10mm/sec CNT100;
   1:  PR[GP1:91,1] = PR[GP1:90,1] + 10.706;
   1:  PR[GP1:91,2] = PR[GP1:90,2] + 39.265;
   1:L PR[91] 10mm/sec CNT100;
   1:  PR[GP1:91,1] = PR[GP1:90,1] + 2.277;
   1:  PR[GP1:91,2] = PR[GP1:90,2] + 36.661;
   1:L PR[91] 10mm/sec CNT100;
   1:  PR[GP1:91,1] = PR[GP1:90,1] + -1.403;
   1:  PR[GP1:91,2] = PR[GP1:90,2] + 37.040;
   1:  PR[GP1:91,3] = PR[GP1:90,3] + 82.460;
   1:L PR[91] 10mm/sec CNT100;
   1:  PR[GP1:91,1] = PR[GP1:90,1] + -9.238;
   1:  PR[GP1:91,2] = PR[GP1:90,2] + 39.459;
   1:L PR[91] 10mm/sec CNT100;
   1:  PR[GP1:91,1] = PR[GP1:90,1] + -14.904;
   1:  PR[GP1:91,2] = PR[GP1:90,2] + 39.662;
   1:L PR[91] 10mm/sec CNT100;
   1:  PR[GP1:91,1] = PR[GP1:90,1] + -24.150;
   1:  PR[GP1:91,2] = PR[GP1:90,2] + 39.493;
   1:L PR[91] 10mm/sec CNT100;
   1:  PR[GP1:91,1] = PR[GP1:90,1] + -28.426;
   1:  PR[GP1:91,2] = PR[GP1:90,2] + 38.091;
   1:L PR[91] 10mm/sec CNT100;
   1:  PR[GP1:91,1] = PR[GP1:90,1] + -37.983;
   1:  PR[GP1:91,2] = PR[GP1:90,2] + 34.564;
   1:L PR[91] 10mm/sec CNT100;
   1:  PR[GP1:91,1] = PR[GP1:90,1] + -40.602;
   1:  PR[GP1:91,2] = PR[GP1:90,2] + 32.491;
   1:L PR[91] 10mm/sec CNT100;
   1:  PR[GP1:91,1] = PR[GP1:90,1] + -49.079;
   1:  PR[GP1:91,2] = PR[GP1:90,2] + 25.494;
   1:L PR[91] 10mm/sec CNT100;
   1:  PR[GP1:91,1] = PR[GP1:90,1] + -50.290;
   1:  PR[GP1:91,2] = PR[GP1:90,2] + 23.491;
   1:L PR[91] 10mm/sec CNT100;
   1:  PR[GP1:91,1] = PR[GP1:90,1] + -56.212;
   1:  PR[GP1:91,2] = PR[GP1:90,2] + 13.472;
   1:L PR[91] 10mm/sec CNT100;
   1:  PR[GP1:91,1] = PR[GP1:90,1] + -58.424;
   1:  PR[GP1:91,2] = PR[GP1:90,2] + 1.266;
   1:L PR[91] 10mm/sec CNT100;
   1:  PR[GP1:91,1] = PR[GP1:90,1] + -58.628;
   1:  PR[GP1:91,2] = PR[GP1:90,2] + 0.002;
   1:L PR[91] 10mm/sec CNT100;
   1:  PR[GP1:91,1] = PR[GP1:90,1] + -56.700;
   1:  PR[GP1:91,2] = PR[GP1:90,2] + -10.592;
   1:L PR[91] 10mm/sec CNT100;
   1:  PR[GP1:91,1] = PR[GP1:90,1] + -56.510;
   1:  PR[GP1:91,2] = PR[GP1:90,2] + -11.862;
   1:L PR[91] 10mm/sec CNT100;
   1:  PR[GP1:91,1] = PR[GP1:90,1] + -56.211;
   1:  PR[GP1:91,2] = PR[GP1:90,2] + -13.483;
   1:L PR[91] 10mm/sec CNT100;
   1:  PR[GP1:91,1] = PR[GP1:90,1] + -50.286;
   1:  PR[GP1:91,2] = PR[GP1:90,2] + -23.505;
   1:L PR[91] 10mm/sec CNT100;
   1:  PR[GP1:91,1] = PR[GP1:90,1] + -49.075;
   1:  PR[GP1:91,2] = PR[GP1:90,2] + -25.509;
   1:L PR[91] 10mm/sec CNT100;
   1:  PR[GP1:91,1] = PR[GP1:90,1] + -40.593;
   1:  PR[GP1:91,2] = PR[GP1:90,2] + -32.505;
   1:L PR[91] 10mm/sec CNT100;
   1:  PR[GP1:91,1] = PR[GP1:90,1] + -37.974;
   1:  PR[GP1:91,2] = PR[GP1:90,2] + -34.578;
   1:L PR[91] 10mm/sec CNT100;
   1:  PR[GP1:91,1] = PR[GP1:90,1] + -28.415;
   1:  PR[GP1:91,2] = PR[GP1:90,2] + -38.101;
   1:L PR[91] 10mm/sec CNT100;
   1:  PR[GP1:91,1] = PR[GP1:90,1] + -24.139;
   1:  PR[GP1:91,2] = PR[GP1:90,2] + -39.504;
   1:L PR[91] 10mm/sec CNT100;
   1:  PR[GP1:91,1] = PR[GP1:90,1] + -14.892;
   1:  PR[GP1:91,2] = PR[GP1:90,2] + -39.668;
   1:L PR[91] 10mm/sec CNT100;
   1:  PR[GP1:91,1] = PR[GP1:90,1] + -9.228;
   1:  PR[GP1:91,2] = PR[GP1:90,2] + -39.466;
   1:L PR[91] 10mm/sec CNT100;
   1:  PR[GP1:91,1] = PR[GP1:90,1] + -1.405;
   1:  PR[GP1:91,2] = PR[GP1:90,2] + -37.033;
   1:L PR[91] 10mm/sec CNT100;
   1:  PR[GP1:91,1] = PR[GP1:90,1] + 2.224;
   1:  PR[GP1:91,2] = PR[GP1:90,2] + -37.032;
   1:L PR[91] 10mm/sec CNT100;
   1:  PR[GP1:91,1] = PR[GP1:90,1] + 10.048;
   1:  PR[GP1:91,2] = PR[GP1:90,2] + -39.466;
   1:L PR[91] 10mm/sec CNT100;
   1:  PR[GP1:91,1] = PR[GP1:90,1] + 15.711;
   1:  PR[GP1:91,2] = PR[GP1:90,2] + -39.668;
   1:L PR[91] 10mm/sec CNT100;
   1:  PR[GP1:91,1] = PR[GP1:90,1] + 24.958;
   1:  PR[GP1:91,2] = PR[GP1:90,2] + -39.505;
   1:L PR[91] 10mm/sec CNT100;
   1:  PR[GP1:91,1] = PR[GP1:90,1] + 29.234;
   1:  PR[GP1:91,2] = PR[GP1:90,2] + -38.102;
   1:L PR[91] 10mm/sec CNT100;
   1:  PR[GP1:91,1] = PR[GP1:90,1] + 38.794;
   1:  PR[GP1:91,2] = PR[GP1:90,2] + -34.580;
   1:L PR[91] 10mm/sec CNT100;
   1:  PR[GP1:91,1] = PR[GP1:90,1] + 41.413;
   1:  PR[GP1:91,2] = PR[GP1:90,2] + -32.507;
   1:L PR[91] 10mm/sec CNT100;
   1:  PR[GP1:91,1] = PR[GP1:90,1] + 49.895;
   1:  PR[GP1:91,2] = PR[GP1:90,2] + -25.503;
   1:L PR[91] 10mm/sec CNT100;
   1:  PR[GP1:91,1] = PR[GP1:90,1] + 51.106;
   1:  PR[GP1:91,2] = PR[GP1:90,2] + -23.500;
   1:L PR[91] 10mm/sec CNT100;
   1:  PR[GP1:91,1] = PR[GP1:90,1] + 57.031;
   1:  PR[GP1:91,2] = PR[GP1:90,2] + -13.500;
   1:L PR[91] 10mm/sec CNT100;
   1:  PR[GP1:91,1] = PR[GP1:90,1] + 59.245;
   1:  PR[GP1:91,2] = PR[GP1:90,2] + -1.276;
   1:L PR[91] 10mm/sec CNT100;
   1:  PR[GP1:91,1] = PR[GP1:90,1] + 59.449;
   1:  PR[GP1:91,2] = PR[GP1:90,2] + -0.011;
   1:L PR[91] 10mm/sec CNT100;
   1:  PR[GP1:91,1] = PR[GP1:90,1] + 57.522;
   1:  PR[GP1:91,2] = PR[GP1:90,2] + 10.595;
   1:L PR[91] 10mm/sec CNT100;
   1:  PR[GP1:91,1] = PR[GP1:90,1] + 57.332;
   1:  PR[GP1:91,2] = PR[GP1:90,2] + 11.866;
   1:L PR[91] 10mm/sec CNT100;
   1:  PR[GP1:91,1] = PR[GP1:90,1] + 57.032;
   1:  PR[GP1:91,2] = PR[GP1:90,2] + 13.487;
   1:L PR[91] 10mm/sec CNT100;
   1:  PR[GP1:91,1] = PR[GP1:90,1] + 51.111;
   1:  PR[GP1:91,2] = PR[GP1:90,2] + 23.486;
   1:L PR[91] 10mm/sec CNT100;
   1:  PR[GP1:91,1] = PR[GP1:90,1] + 49.899;
   1:  PR[GP1:91,2] = PR[GP1:90,2] + 25.489;
   1:L PR[91] 10mm/sec CNT100;
   1:  PR[GP1:91,1] = PR[GP1:90,1] + 41.421;
   1:  PR[GP1:91,2] = PR[GP1:90,2] + 32.494;
   1:L PR[91] 10mm/sec CNT100;
   1:  PR[GP1:91,1] = PR[GP1:90,1] + 38.803;
   1:  PR[GP1:91,2] = PR[GP1:90,2] + 34.567;
   1:L PR[91] 10mm/sec CNT100;
   1:  PR[GP1:91,1] = PR[GP1:90,1] + 29.245;
   1:  PR[GP1:91,2] = PR[GP1:90,2] + 38.091;
   1:L PR[91] 10mm/sec CNT100;
   1:  PR[GP1:91,1] = PR[GP1:90,1] + 24.969;
   1:  PR[GP1:91,2] = PR[GP1:90,2] + 39.494;
   1:L PR[91] 10mm/sec CNT100;
   1:  PR[GP1:91,1] = PR[GP1:90,1] + 15.723;
   1:  PR[GP1:91,2] = PR[GP1:90,2] + 39.661;
   1:L PR[91] 10mm/sec CNT100;
   1:  PR[GP1:91,1] = PR[GP1:90,1] + 10.057;
   1:  PR[GP1:91,2] = PR[GP1:90,2] + 39.458;
   1:L PR[91] 10mm/sec CNT100;
   1:  PR[GP1:91,1] = PR[GP1:90,1] + 2.222;
   1:  PR[GP1:91,2] = PR[GP1:90,2] + 37.039;
   1:L PR[91] 10mm/sec CNT100;
   1:  PR[GP1:91,1] = PR[GP1:90,1] + -1.348;
   1:  PR[GP1:91,2] = PR[GP1:90,2] + 37.418;
   1:  PR[GP1:91,3] = PR[GP1:90,3] + 83.790;
   1:L PR[91] 10mm/sec CNT100;
   1:  PR[GP1:91,1] = PR[GP1:90,1] + -8.589;
   1:  PR[GP1:91,2] = PR[GP1:90,2] + 39.652;
   1:L PR[91] 10mm/sec CNT100;
   1:  PR[GP1:91,1] = PR[GP1:90,1] + -14.987;
   1:  PR[GP1:91,2] = PR[GP1:90,2] + 39.881;
   1:L PR[91] 10mm/sec CNT100;
   1:  PR[GP1:91,1] = PR[GP1:90,1] + -23.580;
   1:  PR[GP1:91,2] = PR[GP1:90,2] + 39.725;
   1:L PR[91] 10mm/sec CNT100;
   1:  PR[GP1:91,1] = PR[GP1:90,1] + -28.575;
   1:  PR[GP1:91,2] = PR[GP1:90,2] + 38.087;
   1:L PR[91] 10mm/sec CNT100;
   1:  PR[GP1:91,1] = PR[GP1:90,1] + -37.500;
   1:  PR[GP1:91,2] = PR[GP1:90,2] + 34.793;
   1:L PR[91] 10mm/sec CNT100;
   1:  PR[GP1:91,1] = PR[GP1:90,1] + -40.732;
   1:  PR[GP1:91,2] = PR[GP1:90,2] + 32.235;
   1:L PR[91] 10mm/sec CNT100;
   1:  PR[GP1:91,1] = PR[GP1:90,1] + -48.677;
   1:  PR[GP1:91,2] = PR[GP1:90,2] + 25.678;
   1:L PR[91] 10mm/sec CNT100;
   1:  PR[GP1:91,1] = PR[GP1:90,1] + -50.306;
   1:  PR[GP1:91,2] = PR[GP1:90,2] + 22.984;
   1:L PR[91] 10mm/sec CNT100;
   1:  PR[GP1:91,1] = PR[GP1:90,1] + -55.866;
   1:  PR[GP1:91,2] = PR[GP1:90,2] + 13.574;
   1:L PR[91] 10mm/sec CNT100;
   1:  PR[GP1:91,1] = PR[GP1:90,1] + -57.944;
   1:  PR[GP1:91,2] = PR[GP1:90,2] + 2.113;
   1:L PR[91] 10mm/sec CNT100;
   1:  PR[GP1:91,1] = PR[GP1:90,1] + -58.284;
   1:  PR[GP1:91,2] = PR[GP1:90,2] + 0.002;
   1:L PR[91] 10mm/sec CNT100;
   1:  PR[GP1:91,1] = PR[GP1:90,1] + -56.594;
   1:  PR[GP1:91,2] = PR[GP1:90,2] + -9.287;
   1:L PR[91] 10mm/sec CNT100;
   1:  PR[GP1:91,1] = PR[GP1:90,1] + -56.314;
   1:  PR[GP1:91,2] = PR[GP1:90,2] + -11.152;
   1:L PR[91] 10mm/sec CNT100;
   1:  PR[GP1:91,1] = PR[GP1:90,1] + -55.865;
   1:  PR[GP1:91,2] = PR[GP1:90,2] + -13.586;
   1:L PR[91] 10mm/sec CNT100;
   1:  PR[GP1:91,1] = PR[GP1:90,1] + -50.301;
   1:  PR[GP1:91,2] = PR[GP1:90,2] + -22.997;
   1:L PR[91] 10mm/sec CNT100;
   1:  PR[GP1:91,1] = PR[GP1:90,1] + -48.672;
   1:  PR[GP1:91,2] = PR[GP1:90,2] + -25.692;
   1:L PR[91] 10mm/sec CNT100;
   1:  PR[GP1:91,1] = PR[GP1:90,1] + -40.724;
   1:  PR[GP1:91,2] = PR[GP1:90,2] + -32.248;
   1:L PR[91] 10mm/sec CNT100;
   1:  PR[GP1:91,1] = PR[GP1:90,1] + -37.492;
   1:  PR[GP1:91,2] = PR[GP1:90,2] + -34.806;
   1:L PR[91] 10mm/sec CNT100;
   1:  PR[GP1:91,1] = PR[GP1:90,1] + -28.565;
   1:  PR[GP1:91,2] = PR[GP1:90,2] + -38.097;
   1:L PR[91] 10mm/sec CNT100;
   1:  PR[GP1:91,1] = PR[GP1:90,1] + -23.570;
   1:  PR[GP1:91,2] = PR[GP1:90,2] + -39.735;
   1:L PR[91] 10mm/sec CNT100;
   1:  PR[GP1:91,1] = PR[GP1:90,1] + -14.976;
   1:  PR[GP1:91,2] = PR[GP1:90,2] + -39.888;
   1:L PR[91] 10mm/sec CNT100;
   1:  PR[GP1:91,1] = PR[GP1:90,1] + -8.581;
   1:  PR[GP1:91,2] = PR[GP1:90,2] + -39.660;
   1:L PR[91] 10mm/sec CNT100;
   1:  PR[GP1:91,1] = PR[GP1:90,1] + -1.350;
   1:  PR[GP1:91,2] = PR[GP1:90,2] + -37.412;
   1:L PR[91] 10mm/sec CNT100;
   1:  PR[GP1:91,1] = PR[GP1:90,1] + 2.169;
   1:  PR[GP1:91,2] = PR[GP1:90,2] + -37.411;
   1:L PR[91] 10mm/sec CNT100;
   1:  PR[GP1:91,1] = PR[GP1:90,1] + 9.401;
   1:  PR[GP1:91,2] = PR[GP1:90,2] + -39.659;
   1:L PR[91] 10mm/sec CNT100;
   1:  PR[GP1:91,1] = PR[GP1:90,1] + 15.796;
   1:  PR[GP1:91,2] = PR[GP1:90,2] + -39.887;
   1:L PR[91] 10mm/sec CNT100;
   1:  PR[GP1:91,1] = PR[GP1:90,1] + 24.390;
   1:  PR[GP1:91,2] = PR[GP1:90,2] + -39.736;
   1:L PR[91] 10mm/sec CNT100;
   1:  PR[GP1:91,1] = PR[GP1:90,1] + 29.384;
   1:  PR[GP1:91,2] = PR[GP1:90,2] + -38.097;
   1:L PR[91] 10mm/sec CNT100;
   1:  PR[GP1:91,1] = PR[GP1:90,1] + 38.312;
   1:  PR[GP1:91,2] = PR[GP1:90,2] + -34.808;
   1:L PR[91] 10mm/sec CNT100;
   1:  PR[GP1:91,1] = PR[GP1:90,1] + 41.544;
   1:  PR[GP1:91,2] = PR[GP1:90,2] + -32.250;
   1:L PR[91] 10mm/sec CNT100;
   1:  PR[GP1:91,1] = PR[GP1:90,1] + 49.493;
   1:  PR[GP1:91,2] = PR[GP1:90,2] + -25.686;
   1:L PR[91] 10mm/sec CNT100;
   1:  PR[GP1:91,1] = PR[GP1:90,1] + 51.122;
   1:  PR[GP1:91,2] = PR[GP1:90,2] + -22.993;
   1:L PR[91] 10mm/sec CNT100;
   1:  PR[GP1:91,1] = PR[GP1:90,1] + 56.685;
   1:  PR[GP1:91,2] = PR[GP1:90,2] + -13.602;
   1:L PR[91] 10mm/sec CNT100;
   1:  PR[GP1:91,1] = PR[GP1:90,1] + 58.765;
   1:  PR[GP1:91,2] = PR[GP1:90,2] + -2.122;
   1:L PR[91] 10mm/sec CNT100;
   1:  PR[GP1:91,1] = PR[GP1:90,1] + 59.105;
   1:  PR[GP1:91,2] = PR[GP1:90,2] + -0.011;
   1:L PR[91] 10mm/sec CNT100;
   1:  PR[GP1:91,1] = PR[GP1:90,1] + 57.415;
   1:  PR[GP1:91,2] = PR[GP1:90,2] + 9.289;
   1:L PR[91] 10mm/sec CNT100;
   1:  PR[GP1:91,1] = PR[GP1:90,1] + 57.136;
   1:  PR[GP1:91,2] = PR[GP1:90,2] + 11.155;
   1:L PR[91] 10mm/sec CNT100;
   1:  PR[GP1:91,1] = PR[GP1:90,1] + 56.687;
   1:  PR[GP1:91,2] = PR[GP1:90,2] + 13.589;
   1:L PR[91] 10mm/sec CNT100;
   1:  PR[GP1:91,1] = PR[GP1:90,1] + 51.126;
   1:  PR[GP1:91,2] = PR[GP1:90,2] + 22.979;
   1:L PR[91] 10mm/sec CNT100;
   1:  PR[GP1:91,1] = PR[GP1:90,1] + 49.497;
   1:  PR[GP1:91,2] = PR[GP1:90,2] + 25.673;
   1:L PR[91] 10mm/sec CNT100;
   1:  PR[GP1:91,1] = PR[GP1:90,1] + 41.552;
   1:  PR[GP1:91,2] = PR[GP1:90,2] + 32.237;
   1:L PR[91] 10mm/sec CNT100;
   1:  PR[GP1:91,1] = PR[GP1:90,1] + 38.320;
   1:  PR[GP1:91,2] = PR[GP1:90,2] + 34.795;
   1:L PR[91] 10mm/sec CNT100;
   1:  PR[GP1:91,1] = PR[GP1:90,1] + 29.394;
   1:  PR[GP1:91,2] = PR[GP1:90,2] + 38.087;
   1:L PR[91] 10mm/sec CNT100;
   1:  PR[GP1:91,1] = PR[GP1:90,1] + 24.400;
   1:  PR[GP1:91,2] = PR[GP1:90,2] + 39.725;
   1:L PR[91] 10mm/sec CNT100;
   1:  PR[GP1:91,1] = PR[GP1:90,1] + 15.807;
   1:  PR[GP1:91,2] = PR[GP1:90,2] + 39.881;
   1:L PR[91] 10mm/sec CNT100;
   1:  PR[GP1:91,1] = PR[GP1:90,1] + 9.409;
   1:  PR[GP1:91,2] = PR[GP1:90,2] + 39.651;
   1:L PR[91] 10mm/sec CNT100;
   1:  PR[GP1:91,1] = PR[GP1:90,1] + 2.167;
   1:  PR[GP1:91,2] = PR[GP1:90,2] + 37.417;
   1:L PR[91] 10mm/sec CNT100;
   1:  PR[GP1:91,1] = PR[GP1:90,1] + -1.293;
   1:  PR[GP1:91,2] = PR[GP1:90,2] + 37.795;
   1:  PR[GP1:91,3] = PR[GP1:90,3] + 85.120;
   1:L PR[91] 10mm/sec CNT100;
   1:  PR[GP1:91,1] = PR[GP1:90,1] + -7.940;
   1:  PR[GP1:91,2] = PR[GP1:90,2] + 39.845;
   1:L PR[91] 10mm/sec CNT100;
   1:  PR[GP1:91,1] = PR[GP1:90,1] + -15.070;
   1:  PR[GP1:91,2] = PR[GP1:90,2] + 40.101;
   1:L PR[91] 10mm/sec CNT100;
   1:  PR[GP1:91,1] = PR[GP1:90,1] + -23.010;
   1:  PR[GP1:91,2] = PR[GP1:90,2] + 39.956;
   1:L PR[91] 10mm/sec CNT100;
   1:  PR[GP1:91,1] = PR[GP1:90,1] + -28.724;
   1:  PR[GP1:91,2] = PR[GP1:90,2] + 38.082;
   1:L PR[91] 10mm/sec CNT100;
   1:  PR[GP1:91,1] = PR[GP1:90,1] + -37.017;
   1:  PR[GP1:91,2] = PR[GP1:90,2] + 35.022;
   1:L PR[91] 10mm/sec CNT100;
   1:  PR[GP1:91,1] = PR[GP1:90,1] + -40.863;
   1:  PR[GP1:91,2] = PR[GP1:90,2] + 31.978;
   1:L PR[91] 10mm/sec CNT100;
   1:  PR[GP1:91,1] = PR[GP1:90,1] + -48.274;
   1:  PR[GP1:91,2] = PR[GP1:90,2] + 25.861;
   1:L PR[91] 10mm/sec CNT100;
   1:  PR[GP1:91,1] = PR[GP1:90,1] + -50.321;
   1:  PR[GP1:91,2] = PR[GP1:90,2] + 22.476;
   1:L PR[91] 10mm/sec CNT100;
   1:  PR[GP1:91,1] = PR[GP1:90,1] + -55.520;
   1:  PR[GP1:91,2] = PR[GP1:90,2] + 13.677;
   1:L PR[91] 10mm/sec CNT100;
   1:  PR[GP1:91,1] = PR[GP1:90,1] + -57.464;
   1:  PR[GP1:91,2] = PR[GP1:90,2] + 2.959;
   1:L PR[91] 10mm/sec CNT100;
   1:  PR[GP1:91,1] = PR[GP1:90,1] + -57.940;
   1:  PR[GP1:91,2] = PR[GP1:90,2] + 0.002;
   1:L PR[91] 10mm/sec CNT100;
   1:  PR[GP1:91,1] = PR[GP1:90,1] + -56.487;
   1:  PR[GP1:91,2] = PR[GP1:90,2] + -7.983;
   1:L PR[91] 10mm/sec CNT100;
   1:  PR[GP1:91,1] = PR[GP1:90,1] + -56.119;
   1:  PR[GP1:91,2] = PR[GP1:90,2] + -10.442;
   1:L PR[91] 10mm/sec CNT100;
   1:  PR[GP1:91,1] = PR[GP1:90,1] + -55.520;
   1:  PR[GP1:91,2] = PR[GP1:90,2] + -13.688;
   1:L PR[91] 10mm/sec CNT100;
   1:  PR[GP1:91,1] = PR[GP1:90,1] + -50.317;
   1:  PR[GP1:91,2] = PR[GP1:90,2] + -22.490;
   1:L PR[91] 10mm/sec CNT100;
   1:  PR[GP1:91,1] = PR[GP1:90,1] + -48.270;
   1:  PR[GP1:91,2] = PR[GP1:90,2] + -25.875;
   1:L PR[91] 10mm/sec CNT100;
   1:  PR[GP1:91,1] = PR[GP1:90,1] + -40.856;
   1:  PR[GP1:91,2] = PR[GP1:90,2] + -31.991;
   1:L PR[91] 10mm/sec CNT100;
   1:  PR[GP1:91,1] = PR[GP1:90,1] + -37.010;
   1:  PR[GP1:91,2] = PR[GP1:90,2] + -35.035;
   1:L PR[91] 10mm/sec CNT100;
   1:  PR[GP1:91,1] = PR[GP1:90,1] + -28.715;
   1:  PR[GP1:91,2] = PR[GP1:90,2] + -38.092;
   1:L PR[91] 10mm/sec CNT100;
   1:  PR[GP1:91,1] = PR[GP1:90,1] + -23.001;
   1:  PR[GP1:91,2] = PR[GP1:90,2] + -39.967;
   1:L PR[91] 10mm/sec CNT100;
   1:  PR[GP1:91,1] = PR[GP1:90,1] + -15.061;
   1:  PR[GP1:91,2] = PR[GP1:90,2] + -40.108;
   1:L PR[91] 10mm/sec CNT100;
   1:  PR[GP1:91,1] = PR[GP1:90,1] + -7.933;
   1:  PR[GP1:91,2] = PR[GP1:90,2] + -39.853;
   1:L PR[91] 10mm/sec CNT100;
   1:  PR[GP1:91,1] = PR[GP1:90,1] + -1.295;
   1:  PR[GP1:91,2] = PR[GP1:90,2] + -37.791;
   1:L PR[91] 10mm/sec CNT100;
   1:  PR[GP1:91,1] = PR[GP1:90,1] + 2.114;
   1:  PR[GP1:91,2] = PR[GP1:90,2] + -37.790;
   1:L PR[91] 10mm/sec CNT100;
   1:  PR[GP1:91,1] = PR[GP1:90,1] + 8.753;
   1:  PR[GP1:91,2] = PR[GP1:90,2] + -39.853;
   1:L PR[91] 10mm/sec CNT100;
   1:  PR[GP1:91,1] = PR[GP1:90,1] + 15.881;
   1:  PR[GP1:91,2] = PR[GP1:90,2] + -40.107;
   1:L PR[91] 10mm/sec CNT100;
   1:  PR[GP1:91,1] = PR[GP1:90,1] + 23.821;
   1:  PR[GP1:91,2] = PR[GP1:90,2] + -39.967;
   1:L PR[91] 10mm/sec CNT100;
   1:  PR[GP1:91,1] = PR[GP1:90,1] + 29.534;
   1:  PR[GP1:91,2] = PR[GP1:90,2] + -38.093;
   1:L PR[91] 10mm/sec CNT100;
   1:  PR[GP1:91,1] = PR[GP1:90,1] + 37.830;
   1:  PR[GP1:91,2] = PR[GP1:90,2] + -35.037;
   1:L PR[91] 10mm/sec CNT100;
   1:  PR[GP1:91,1] = PR[GP1:90,1] + 41.675;
   1:  PR[GP1:91,2] = PR[GP1:90,2] + -31.993;
   1:L PR[91] 10mm/sec CNT100;
   1:  PR[GP1:91,1] = PR[GP1:90,1] + 49.090;
   1:  PR[GP1:91,2] = PR[GP1:90,2] + -25.870;
   1:L PR[91] 10mm/sec CNT100;
   1:  PR[GP1:91,1] = PR[GP1:90,1] + 51.137;
   1:  PR[GP1:91,2] = PR[GP1:90,2] + -22.486;
   1:L PR[91] 10mm/sec CNT100;
   1:  PR[GP1:91,1] = PR[GP1:90,1] + 56.340;
   1:  PR[GP1:91,2] = PR[GP1:90,2] + -13.704;
   1:L PR[91] 10mm/sec CNT100;
   1:  PR[GP1:91,1] = PR[GP1:90,1] + 58.284;
   1:  PR[GP1:91,2] = PR[GP1:90,2] + -2.969;
   1:L PR[91] 10mm/sec CNT100;
   1:  PR[GP1:91,1] = PR[GP1:90,1] + 58.761;
   1:  PR[GP1:91,2] = PR[GP1:90,2] + -0.011;
   1:L PR[91] 10mm/sec CNT100;
   1:  PR[GP1:91,1] = PR[GP1:90,1] + 57.308;
   1:  PR[GP1:91,2] = PR[GP1:90,2] + 7.983;
   1:L PR[91] 10mm/sec CNT100;
   1:  PR[GP1:91,1] = PR[GP1:90,1] + 56.940;
   1:  PR[GP1:91,2] = PR[GP1:90,2] + 10.444;
   1:L PR[91] 10mm/sec CNT100;
   1:  PR[GP1:91,1] = PR[GP1:90,1] + 56.341;
   1:  PR[GP1:91,2] = PR[GP1:90,2] + 13.692;
   1:L PR[91] 10mm/sec CNT100;
   1:  PR[GP1:91,1] = PR[GP1:90,1] + 51.141;
   1:  PR[GP1:91,2] = PR[GP1:90,2] + 22.472;
   1:L PR[91] 10mm/sec CNT100;
   1:  PR[GP1:91,1] = PR[GP1:90,1] + 49.094;
   1:  PR[GP1:91,2] = PR[GP1:90,2] + 25.856;
   1:L PR[91] 10mm/sec CNT100;
   1:  PR[GP1:91,1] = PR[GP1:90,1] + 41.682;
   1:  PR[GP1:91,2] = PR[GP1:90,2] + 31.980;
   1:L PR[91] 10mm/sec CNT100;
   1:  PR[GP1:91,1] = PR[GP1:90,1] + 37.837;
   1:  PR[GP1:91,2] = PR[GP1:90,2] + 35.024;
   1:L PR[91] 10mm/sec CNT100;
   1:  PR[GP1:91,1] = PR[GP1:90,1] + 29.543;
   1:  PR[GP1:91,2] = PR[GP1:90,2] + 38.083;
   1:L PR[91] 10mm/sec CNT100;
   1:  PR[GP1:91,1] = PR[GP1:90,1] + 23.830;
   1:  PR[GP1:91,2] = PR[GP1:90,2] + 39.956;
   1:L PR[91] 10mm/sec CNT100;
   1:  PR[GP1:91,1] = PR[GP1:90,1] + 15.890;
   1:  PR[GP1:91,2] = PR[GP1:90,2] + 40.100;
   1:L PR[91] 10mm/sec CNT100;
   1:  PR[GP1:91,1] = PR[GP1:90,1] + 8.760;
   1:  PR[GP1:91,2] = PR[GP1:90,2] + 39.845;
   1:L PR[91] 10mm/sec CNT100;
   1:  PR[GP1:91,1] = PR[GP1:90,1] + 2.113;
   1:  PR[GP1:91,2] = PR[GP1:90,2] + 37.794;
   1:L PR[91] 10mm/sec CNT100;
   1:  PR[GP1:91,1] = PR[GP1:90,1] + -1.238;
   1:  PR[GP1:91,2] = PR[GP1:90,2] + 38.173;
   1:  PR[GP1:91,3] = PR[GP1:90,3] + 86.450;
   1:L PR[91] 10mm/sec CNT100;
   1:  PR[GP1:91,1] = PR[GP1:90,1] + -7.291;
   1:  PR[GP1:91,2] = PR[GP1:90,2] + 40.039;
   1:L PR[91] 10mm/sec CNT100;
   1:  PR[GP1:91,1] = PR[GP1:90,1] + -15.154;
   1:  PR[GP1:91,2] = PR[GP1:90,2] + 40.320;
   1:L PR[91] 10mm/sec CNT100;
   1:  PR[GP1:91,1] = PR[GP1:90,1] + -22.440;
   1:  PR[GP1:91,2] = PR[GP1:90,2] + 40.187;
   1:L PR[91] 10mm/sec CNT100;
   1:  PR[GP1:91,1] = PR[GP1:90,1] + -28.873;
   1:  PR[GP1:91,2] = PR[GP1:90,2] + 38.078;
   1:L PR[91] 10mm/sec CNT100;
   1:  PR[GP1:91,1] = PR[GP1:90,1] + -36.534;
   1:  PR[GP1:91,2] = PR[GP1:90,2] + 35.251;
   1:L PR[91] 10mm/sec CNT100;
   1:  PR[GP1:91,1] = PR[GP1:90,1] + -40.993;
   1:  PR[GP1:91,2] = PR[GP1:90,2] + 31.722;
   1:L PR[91] 10mm/sec CNT100;
   1:  PR[GP1:91,1] = PR[GP1:90,1] + -47.871;
   1:  PR[GP1:91,2] = PR[GP1:90,2] + 26.045;
   1:L PR[91] 10mm/sec CNT100;
   1:  PR[GP1:91,1] = PR[GP1:90,1] + -50.336;
   1:  PR[GP1:91,2] = PR[GP1:90,2] + 21.969;
   1:L PR[91] 10mm/sec CNT100;
   1:  PR[GP1:91,1] = PR[GP1:90,1] + -55.175;
   1:  PR[GP1:91,2] = PR[GP1:90,2] + 13.780;
   1:L PR[91] 10mm/sec CNT100;
   1:  PR[GP1:91,1] = PR[GP1:90,1] + -56.983;
   1:  PR[GP1:91,2] = PR[GP1:90,2] + 3.805;
   1:L PR[91] 10mm/sec CNT100;
   1:  PR[GP1:91,1] = PR[GP1:90,1] + -57.596;
   1:  PR[GP1:91,2] = PR[GP1:90,2] + 0.002;
   1:L PR[91] 10mm/sec CNT100;
   1:  PR[GP1:91,1] = PR[GP1:90,1] + -56.381;
   1:  PR[GP1:91,2] = PR[GP1:90,2] + -6.678;
   1:L PR[91] 10mm/sec CNT100;
   1:  PR[GP1:91,1] = PR[GP1:90,1] + -55.923;
   1:  PR[GP1:91,2] = PR[GP1:90,2] + -9.732;
   1:L PR[91] 10mm/sec CNT100;
   1:  PR[GP1:91,1] = PR[GP1:90,1] + -55.174;
   1:  PR[GP1:91,2] = PR[GP1:90,2] + -13.791;
   1:L PR[91] 10mm/sec CNT100;
   1:  PR[GP1:91,1] = PR[GP1:90,1] + -50.332;
   1:  PR[GP1:91,2] = PR[GP1:90,2] + -21.982;
   1:L PR[91] 10mm/sec CNT100;
   1:  PR[GP1:91,1] = PR[GP1:90,1] + -47.868;
   1:  PR[GP1:91,2] = PR[GP1:90,2] + -26.058;
   1:L PR[91] 10mm/sec CNT100;
   1:  PR[GP1:91,1] = PR[GP1:90,1] + -40.987;
   1:  PR[GP1:91,2] = PR[GP1:90,2] + -31.734;
   1:L PR[91] 10mm/sec CNT100;
   1:  PR[GP1:91,1] = PR[GP1:90,1] + -36.528;
   1:  PR[GP1:91,2] = PR[GP1:90,2] + -35.263;
   1:L PR[91] 10mm/sec CNT100;
   1:  PR[GP1:91,1] = PR[GP1:90,1] + -28.865;
   1:  PR[GP1:91,2] = PR[GP1:90,2] + -38.088;
   1:L PR[91] 10mm/sec CNT100;
   1:  PR[GP1:91,1] = PR[GP1:90,1] + -22.432;
   1:  PR[GP1:91,2] = PR[GP1:90,2] + -40.198;
   1:L PR[91] 10mm/sec CNT100;
   1:  PR[GP1:91,1] = PR[GP1:90,1] + -15.145;
   1:  PR[GP1:91,2] = PR[GP1:90,2] + -40.327;
   1:L PR[91] 10mm/sec CNT100;
   1:  PR[GP1:91,1] = PR[GP1:90,1] + -7.286;
   1:  PR[GP1:91,2] = PR[GP1:90,2] + -40.047;
   1:L PR[91] 10mm/sec CNT100;
   1:  PR[GP1:91,1] = PR[GP1:90,1] + -1.240;
   1:  PR[GP1:91,2] = PR[GP1:90,2] + -38.170;
   1:L PR[91] 10mm/sec CNT100;
   1:  PR[GP1:91,1] = PR[GP1:90,1] + 2.060;
   1:  PR[GP1:91,2] = PR[GP1:90,2] + -38.169;
   1:L PR[91] 10mm/sec CNT100;
   1:  PR[GP1:91,1] = PR[GP1:90,1] + 8.106;
   1:  PR[GP1:91,2] = PR[GP1:90,2] + -40.047;
   1:L PR[91] 10mm/sec CNT100;
   1:  PR[GP1:91,1] = PR[GP1:90,1] + 15.965;
   1:  PR[GP1:91,2] = PR[GP1:90,2] + -40.327;
   1:L PR[91] 10mm/sec CNT100;
   1:  PR[GP1:91,1] = PR[GP1:90,1] + 23.253;
   1:  PR[GP1:91,2] = PR[GP1:90,2] + -40.198;
   1:L PR[91] 10mm/sec CNT100;
   1:  PR[GP1:91,1] = PR[GP1:90,1] + 29.685;
   1:  PR[GP1:91,2] = PR[GP1:90,2] + -38.088;
   1:L PR[91] 10mm/sec CNT100;
   1:  PR[GP1:91,1] = PR[GP1:90,1] + 37.348;
   1:  PR[GP1:91,2] = PR[GP1:90,2] + -35.265;
   1:L PR[91] 10mm/sec CNT100;
   1:  PR[GP1:91,1] = PR[GP1:90,1] + 41.807;
   1:  PR[GP1:91,2] = PR[GP1:90,2] + -31.735;
   1:L PR[91] 10mm/sec CNT100;
   1:  PR[GP1:91,1] = PR[GP1:90,1] + 48.688;
   1:  PR[GP1:91,2] = PR[GP1:90,2] + -26.053;
   1:L PR[91] 10mm/sec CNT100;
   1:  PR[GP1:91,1] = PR[GP1:90,1] + 51.153;
   1:  PR[GP1:91,2] = PR[GP1:90,2] + -21.978;
   1:L PR[91] 10mm/sec CNT100;
   1:  PR[GP1:91,1] = PR[GP1:90,1] + 55.994;
   1:  PR[GP1:91,2] = PR[GP1:90,2] + -13.806;
   1:L PR[91] 10mm/sec CNT100;
   1:  PR[GP1:91,1] = PR[GP1:90,1] + 57.804;
   1:  PR[GP1:91,2] = PR[GP1:90,2] + -3.815;
   1:L PR[91] 10mm/sec CNT100;
   1:  PR[GP1:91,1] = PR[GP1:90,1] + 58.417;
   1:  PR[GP1:91,2] = PR[GP1:90,2] + -0.011;
   1:L PR[91] 10mm/sec CNT100;
   1:  PR[GP1:91,1] = PR[GP1:90,1] + 57.202;
   1:  PR[GP1:91,2] = PR[GP1:90,2] + 6.676;
   1:L PR[91] 10mm/sec CNT100;
   1:  PR[GP1:91,1] = PR[GP1:90,1] + 56.745;
   1:  PR[GP1:91,2] = PR[GP1:90,2] + 9.734;
   1:L PR[91] 10mm/sec CNT100;
   1:  PR[GP1:91,1] = PR[GP1:90,1] + 55.996;
   1:  PR[GP1:91,2] = PR[GP1:90,2] + 13.794;
   1:L PR[91] 10mm/sec CNT100;
   1:  PR[GP1:91,1] = PR[GP1:90,1] + 51.156;
   1:  PR[GP1:91,2] = PR[GP1:90,2] + 21.965;
   1:L PR[91] 10mm/sec CNT100;
   1:  PR[GP1:91,1] = PR[GP1:90,1] + 48.692;
   1:  PR[GP1:91,2] = PR[GP1:90,2] + 26.040;
   1:L PR[91] 10mm/sec CNT100;
   1:  PR[GP1:91,1] = PR[GP1:90,1] + 41.813;
   1:  PR[GP1:91,2] = PR[GP1:90,2] + 31.723;
   1:L PR[91] 10mm/sec CNT100;
   1:  PR[GP1:91,1] = PR[GP1:90,1] + 37.354;
   1:  PR[GP1:91,2] = PR[GP1:90,2] + 35.253;
   1:L PR[91] 10mm/sec CNT100;
   1:  PR[GP1:91,1] = PR[GP1:90,1] + 29.693;
   1:  PR[GP1:91,2] = PR[GP1:90,2] + 38.078;
   1:L PR[91] 10mm/sec CNT100;
   1:  PR[GP1:91,1] = PR[GP1:90,1] + 23.261;
   1:  PR[GP1:91,2] = PR[GP1:90,2] + 40.188;
   1:L PR[91] 10mm/sec CNT100;
   1:  PR[GP1:91,1] = PR[GP1:90,1] + 15.974;
   1:  PR[GP1:91,2] = PR[GP1:90,2] + 40.320;
   1:L PR[91] 10mm/sec CNT100;
   1:  PR[GP1:91,1] = PR[GP1:90,1] + 8.112;
   1:  PR[GP1:91,2] = PR[GP1:90,2] + 40.038;
   1:L PR[91] 10mm/sec CNT100;
   1:  PR[GP1:91,1] = PR[GP1:90,1] + 2.058;
   1:  PR[GP1:91,2] = PR[GP1:90,2] + 38.172;
   1:L PR[91] 10mm/sec CNT100;
   1:  PR[GP1:91,1] = PR[GP1:90,1] + -1.183;
   1:  PR[GP1:91,2] = PR[GP1:90,2] + 38.551;
   1:  PR[GP1:91,3] = PR[GP1:90,3] + 87.780;
   1:L PR[91] 10mm/sec CNT100;
   1:  PR[GP1:91,1] = PR[GP1:90,1] + -6.642;
   1:  PR[GP1:91,2] = PR[GP1:90,2] + 40.232;
   1:L PR[91] 10mm/sec CNT100;
   1:  PR[GP1:91,1] = PR[GP1:90,1] + -15.237;
   1:  PR[GP1:91,2] = PR[GP1:90,2] + 40.540;
   1:L PR[91] 10mm/sec CNT100;
   1:  PR[GP1:91,1] = PR[GP1:90,1] + -21.871;
   1:  PR[GP1:91,2] = PR[GP1:90,2] + 40.419;
   1:L PR[91] 10mm/sec CNT100;
   1:  PR[GP1:91,1] = PR[GP1:90,1] + -29.022;
   1:  PR[GP1:91,2] = PR[GP1:90,2] + 38.074;
   1:L PR[91] 10mm/sec CNT100;
   1:  PR[GP1:91,1] = PR[GP1:90,1] + -36.051;
   1:  PR[GP1:91,2] = PR[GP1:90,2] + 35.480;
   1:L PR[91] 10mm/sec CNT100;
   1:  PR[GP1:91,1] = PR[GP1:90,1] + -41.124;
   1:  PR[GP1:91,2] = PR[GP1:90,2] + 31.465;
   1:L PR[91] 10mm/sec CNT100;
   1:  PR[GP1:91,1] = PR[GP1:90,1] + -47.469;
   1:  PR[GP1:91,2] = PR[GP1:90,2] + 26.228;
   1:L PR[91] 10mm/sec CNT100;
   1:  PR[GP1:91,1] = PR[GP1:90,1] + -50.351;
   1:  PR[GP1:91,2] = PR[GP1:90,2] + 21.461;
   1:L PR[91] 10mm/sec CNT100;
   1:  PR[GP1:91,1] = PR[GP1:90,1] + -54.829;
   1:  PR[GP1:91,2] = PR[GP1:90,2] + 13.883;
   1:L PR[91] 10mm/sec CNT100;
   1:  PR[GP1:91,1] = PR[GP1:90,1] + -56.503;
   1:  PR[GP1:91,2] = PR[GP1:90,2] + 4.651;
   1:L PR[91] 10mm/sec CNT100;
   1:  PR[GP1:91,1] = PR[GP1:90,1] + -57.252;
   1:  PR[GP1:91,2] = PR[GP1:90,2] + 0.002;
   1:L PR[91] 10mm/sec CNT100;
   1:  PR[GP1:91,1] = PR[GP1:90,1] + -56.274;
   1:  PR[GP1:91,2] = PR[GP1:90,2] + -5.373;
   1:L PR[91] 10mm/sec CNT100;
   1:  PR[GP1:91,1] = PR[GP1:90,1] + -55.728;
   1:  PR[GP1:91,2] = PR[GP1:90,2] + -9.022;
   1:L PR[91] 10mm/sec CNT100;
   1:  PR[GP1:91,1] = PR[GP1:90,1] + -54.829;
   1:  PR[GP1:91,2] = PR[GP1:90,2] + -13.894;
   1:L PR[91] 10mm/sec CNT100;
   1:  PR[GP1:91,1] = PR[GP1:90,1] + -50.348;
   1:  PR[GP1:91,2] = PR[GP1:90,2] + -21.474;
   1:L PR[91] 10mm/sec CNT100;
   1:  PR[GP1:91,1] = PR[GP1:90,1] + -47.466;
   1:  PR[GP1:91,2] = PR[GP1:90,2] + -26.241;
   1:L PR[91] 10mm/sec CNT100;
   1:  PR[GP1:91,1] = PR[GP1:90,1] + -41.118;
   1:  PR[GP1:91,2] = PR[GP1:90,2] + -31.477;
   1:L PR[91] 10mm/sec CNT100;
   1:  PR[GP1:91,1] = PR[GP1:90,1] + -36.045;
   1:  PR[GP1:91,2] = PR[GP1:90,2] + -35.492;
   1:L PR[91] 10mm/sec CNT100;
   1:  PR[GP1:91,1] = PR[GP1:90,1] + -29.015;
   1:  PR[GP1:91,2] = PR[GP1:90,2] + -38.083;
   1:L PR[91] 10mm/sec CNT100;
   1:  PR[GP1:91,1] = PR[GP1:90,1] + -21.864;
   1:  PR[GP1:91,2] = PR[GP1:90,2] + -40.429;
   1:L PR[91] 10mm/sec CNT100;
   1:  PR[GP1:91,1] = PR[GP1:90,1] + -15.229;
   1:  PR[GP1:91,2] = PR[GP1:90,2] + -40.547;
   1:L PR[91] 10mm/sec CNT100;
   1:  PR[GP1:91,1] = PR[GP1:90,1] + -6.638;
   1:  PR[GP1:91,2] = PR[GP1:90,2] + -40.241;
   1:L PR[91] 10mm/sec CNT100;
   1:  PR[GP1:91,1] = PR[GP1:90,1] + -1.185;
   1:  PR[GP1:91,2] = PR[GP1:90,2] + -38.548;
   1:L PR[91] 10mm/sec CNT100;
   1:  PR[GP1:91,1] = PR[GP1:90,1] + 2.005;
   1:L PR[91] 10mm/sec CNT100;
   1:  PR[GP1:91,1] = PR[GP1:90,1] + 7.459;
   1:  PR[GP1:91,2] = PR[GP1:90,2] + -40.240;
   1:L PR[91] 10mm/sec CNT100;
   1:  PR[GP1:91,1] = PR[GP1:90,1] + 16.050;
   1:  PR[GP1:91,2] = PR[GP1:90,2] + -40.546;
   1:L PR[91] 10mm/sec CNT100;
   1:  PR[GP1:91,1] = PR[GP1:90,1] + 22.684;
   1:  PR[GP1:91,2] = PR[GP1:90,2] + -40.429;
   1:L PR[91] 10mm/sec CNT100;
   1:  PR[GP1:91,1] = PR[GP1:90,1] + 29.835;
   1:  PR[GP1:91,2] = PR[GP1:90,2] + -38.083;
   1:L PR[91] 10mm/sec CNT100;
   1:  PR[GP1:91,1] = PR[GP1:90,1] + 36.866;
   1:  PR[GP1:91,2] = PR[GP1:90,2] + -35.493;
   1:L PR[91] 10mm/sec CNT100;
   1:  PR[GP1:91,1] = PR[GP1:90,1] + 41.938;
   1:  PR[GP1:91,2] = PR[GP1:90,2] + -31.478;
   1:L PR[91] 10mm/sec CNT100;
   1:  PR[GP1:91,1] = PR[GP1:90,1] + 48.286;
   1:  PR[GP1:91,2] = PR[GP1:90,2] + -26.236;
   1:L PR[91] 10mm/sec CNT100;
   1:  PR[GP1:91,1] = PR[GP1:90,1] + 51.168;
   1:  PR[GP1:91,2] = PR[GP1:90,2] + -21.471;
   1:L PR[91] 10mm/sec CNT100;
   1:  PR[GP1:91,1] = PR[GP1:90,1] + 55.649;
   1:  PR[GP1:91,2] = PR[GP1:90,2] + -13.908;
   1:L PR[91] 10mm/sec CNT100;
   1:  PR[GP1:91,1] = PR[GP1:90,1] + 57.324;
   1:  PR[GP1:91,2] = PR[GP1:90,2] + -4.661;
   1:L PR[91] 10mm/sec CNT100;
   1:  PR[GP1:91,1] = PR[GP1:90,1] + 58.073;
   1:  PR[GP1:91,2] = PR[GP1:90,2] + -0.011;
   1:L PR[91] 10mm/sec CNT100;
   1:  PR[GP1:91,1] = PR[GP1:90,1] + 57.095;
   1:  PR[GP1:91,2] = PR[GP1:90,2] + 5.370;
   1:L PR[91] 10mm/sec CNT100;
   1:  PR[GP1:91,1] = PR[GP1:90,1] + 56.549;
   1:  PR[GP1:91,2] = PR[GP1:90,2] + 9.023;
   1:L PR[91] 10mm/sec CNT100;
   1:  PR[GP1:91,1] = PR[GP1:90,1] + 55.650;
   1:  PR[GP1:91,2] = PR[GP1:90,2] + 13.896;
   1:L PR[91] 10mm/sec CNT100;
   1:  PR[GP1:91,1] = PR[GP1:90,1] + 51.172;
   1:  PR[GP1:91,2] = PR[GP1:90,2] + 21.459;
   1:L PR[91] 10mm/sec CNT100;
   1:  PR[GP1:91,1] = PR[GP1:90,1] + 48.289;
   1:  PR[GP1:91,2] = PR[GP1:90,2] + 26.224;
   1:L PR[91] 10mm/sec CNT100;
   1:  PR[GP1:91,1] = PR[GP1:90,1] + 41.943;
   1:  PR[GP1:91,2] = PR[GP1:90,2] + 31.466;
   1:L PR[91] 10mm/sec CNT100;
   1:  PR[GP1:91,1] = PR[GP1:90,1] + 36.871;
   1:  PR[GP1:91,2] = PR[GP1:90,2] + 35.481;
   1:L PR[91] 10mm/sec CNT100;
   1:  PR[GP1:91,1] = PR[GP1:90,1] + 29.842;
   1:  PR[GP1:91,2] = PR[GP1:90,2] + 38.074;
   1:L PR[91] 10mm/sec CNT100;
   1:  PR[GP1:91,1] = PR[GP1:90,1] + 22.691;
   1:  PR[GP1:91,2] = PR[GP1:90,2] + 40.419;
   1:L PR[91] 10mm/sec CNT100;
   1:  PR[GP1:91,1] = PR[GP1:90,1] + 16.057;
   1:  PR[GP1:91,2] = PR[GP1:90,2] + 40.539;
   1:L PR[91] 10mm/sec CNT100;
   1:  PR[GP1:91,1] = PR[GP1:90,1] + 7.463;
   1:  PR[GP1:91,2] = PR[GP1:90,2] + 40.231;
   1:L PR[91] 10mm/sec CNT100;
   1:  PR[GP1:91,1] = PR[GP1:90,1] + 2.003;
   1:  PR[GP1:91,2] = PR[GP1:90,2] + 38.550;
   1:L PR[91] 10mm/sec CNT100;
   1:  PR[GP1:91,1] = PR[GP1:90,1] + -1.127;
   1:  PR[GP1:91,2] = PR[GP1:90,2] + 38.928;
   1:  PR[GP1:91,3] = PR[GP1:90,3] + 89.110;
   1:L PR[91] 10mm/sec CNT100;
   1:  PR[GP1:91,1] = PR[GP1:90,1] + -5.993;
   1:  PR[GP1:91,2] = PR[GP1:90,2] + 40.425;
   1:L PR[91] 10mm/sec CNT100;
   1:  PR[GP1:91,1] = PR[GP1:90,1] + -15.320;
   1:  PR[GP1:91,2] = PR[GP1:90,2] + 40.759;
   1:L PR[91] 10mm/sec CNT100;
   1:  PR[GP1:91,1] = PR[GP1:90,1] + -21.301;
   1:  PR[GP1:91,2] = PR[GP1:90,2] + 40.650;
   1:L PR[91] 10mm/sec CNT100;
   1:  PR[GP1:91,1] = PR[GP1:90,1] + -29.171;
   1:  PR[GP1:91,2] = PR[GP1:90,2] + 38.069;
   1:L PR[91] 10mm/sec CNT100;
   1:  PR[GP1:91,1] = PR[GP1:90,1] + -35.568;
   1:  PR[GP1:91,2] = PR[GP1:90,2] + 35.709;
   1:L PR[91] 10mm/sec CNT100;
   1:  PR[GP1:91,1] = PR[GP1:90,1] + -41.254;
   1:  PR[GP1:91,2] = PR[GP1:90,2] + 31.209;
   1:L PR[91] 10mm/sec CNT100;
   1:  PR[GP1:91,1] = PR[GP1:90,1] + -47.066;
   1:  PR[GP1:91,2] = PR[GP1:90,2] + 26.412;
   1:L PR[91] 10mm/sec CNT100;
   1:  PR[GP1:91,1] = PR[GP1:90,1] + -50.366;
   1:  PR[GP1:91,2] = PR[GP1:90,2] + 20.954;
   1:L PR[91] 10mm/sec CNT100;
   1:  PR[GP1:91,1] = PR[GP1:90,1] + -54.484;
   1:  PR[GP1:91,2] = PR[GP1:90,2] + 13.986;
   1:L PR[91] 10mm/sec CNT100;
   1:  PR[GP1:91,1] = PR[GP1:90,1] + -56.023;
   1:  PR[GP1:91,2] = PR[GP1:90,2] + 5.498;
   1:L PR[91] 10mm/sec CNT100;
   1:  PR[GP1:91,1] = PR[GP1:90,1] + -56.908;
   1:  PR[GP1:91,2] = PR[GP1:90,2] + 0.002;
   1:L PR[91] 10mm/sec CNT100;
   1:  PR[GP1:91,1] = PR[GP1:90,1] + -56.168;
   1:  PR[GP1:91,2] = PR[GP1:90,2] + -4.069;
   1:L PR[91] 10mm/sec CNT100;
   1:  PR[GP1:91,1] = PR[GP1:90,1] + -55.532;
   1:  PR[GP1:91,2] = PR[GP1:90,2] + -8.312;
   1:L PR[91] 10mm/sec CNT100;
   1:  PR[GP1:91,1] = PR[GP1:90,1] + -54.483;
   1:  PR[GP1:91,2] = PR[GP1:90,2] + -13.996;
   1:L PR[91] 10mm/sec CNT100;
   1:  PR[GP1:91,1] = PR[GP1:90,1] + -50.363;
   1:  PR[GP1:91,2] = PR[GP1:90,2] + -20.966;
   1:L PR[91] 10mm/sec CNT100;
   1:  PR[GP1:91,1] = PR[GP1:90,1] + -47.063;
   1:  PR[GP1:91,2] = PR[GP1:90,2] + -26.424;
   1:L PR[91] 10mm/sec CNT100;
   1:  PR[GP1:91,1] = PR[GP1:90,1] + -41.249;
   1:  PR[GP1:91,2] = PR[GP1:90,2] + -31.220;
   1:L PR[91] 10mm/sec CNT100;
   1:  PR[GP1:91,1] = PR[GP1:90,1] + -35.563;
   1:  PR[GP1:91,2] = PR[GP1:90,2] + -35.720;
   1:L PR[91] 10mm/sec CNT100;
   1:  PR[GP1:91,1] = PR[GP1:90,1] + -29.165;
   1:  PR[GP1:91,2] = PR[GP1:90,2] + -38.078;
   1:L PR[91] 10mm/sec CNT100;
   1:  PR[GP1:91,1] = PR[GP1:90,1] + -21.295;
   1:  PR[GP1:91,2] = PR[GP1:90,2] + -40.660;
   1:L PR[91] 10mm/sec CNT100;
   1:  PR[GP1:91,1] = PR[GP1:90,1] + -15.314;
   1:  PR[GP1:91,2] = PR[GP1:90,2] + -40.767;
   1:L PR[91] 10mm/sec CNT100;
   1:  PR[GP1:91,1] = PR[GP1:90,1] + -5.991;
   1:  PR[GP1:91,2] = PR[GP1:90,2] + -40.434;
   1:L PR[91] 10mm/sec CNT100;
   1:  PR[GP1:91,1] = PR[GP1:90,1] + -1.129;
   1:  PR[GP1:91,2] = PR[GP1:90,2] + -38.927;
   1:L PR[91] 10mm/sec CNT100;
   1:  PR[GP1:91,1] = PR[GP1:90,1] + 1.950;
   1:  PR[GP1:91,2] = PR[GP1:90,2] + -38.926;
   1:L PR[91] 10mm/sec CNT100;
   1:  PR[GP1:91,1] = PR[GP1:90,1] + 6.812;
   1:  PR[GP1:91,2] = PR[GP1:90,2] + -40.434;
   1:L PR[91] 10mm/sec CNT100;
   1:  PR[GP1:91,1] = PR[GP1:90,1] + 16.134;
   1:  PR[GP1:91,2] = PR[GP1:90,2] + -40.766;
   1:L PR[91] 10mm/sec CNT100;
   1:  PR[GP1:91,1] = PR[GP1:90,1] + 22.116;
   1:  PR[GP1:91,2] = PR[GP1:90,2] + -40.661;
   1:L PR[91] 10mm/sec CNT100;
   1:  PR[GP1:91,1] = PR[GP1:90,1] + 29.985;
   1:  PR[GP1:91,2] = PR[GP1:90,2] + -38.079;
   1:L PR[91] 10mm/sec CNT100;
   1:  PR[GP1:91,1] = PR[GP1:90,1] + 36.384;
   1:  PR[GP1:91,2] = PR[GP1:90,2] + -35.722;
   1:L PR[91] 10mm/sec CNT100;
   1:  PR[GP1:91,1] = PR[GP1:90,1] + 42.069;
   1:  PR[GP1:91,2] = PR[GP1:90,2] + -31.221;
   1:L PR[91] 10mm/sec CNT100;
   1:  PR[GP1:91,1] = PR[GP1:90,1] + 47.884;
   1:  PR[GP1:91,2] = PR[GP1:90,2] + -26.419;
   1:L PR[91] 10mm/sec CNT100;
   1:  PR[GP1:91,1] = PR[GP1:90,1] + 51.184;
   1:  PR[GP1:91,2] = PR[GP1:90,2] + -20.964;
   1:L PR[91] 10mm/sec CNT100;
   1:  PR[GP1:91,1] = PR[GP1:90,1] + 55.303;
   1:  PR[GP1:91,2] = PR[GP1:90,2] + -14.010;
   1:L PR[91] 10mm/sec CNT100;
   1:  PR[GP1:91,1] = PR[GP1:90,1] + 56.843;
   1:  PR[GP1:91,2] = PR[GP1:90,2] + -5.508;
   1:L PR[91] 10mm/sec CNT100;
   1:  PR[GP1:91,1] = PR[GP1:90,1] + 57.729;
   1:  PR[GP1:91,2] = PR[GP1:90,2] + -0.011;
   1:L PR[91] 10mm/sec CNT100;
   1:  PR[GP1:91,1] = PR[GP1:90,1] + 56.989;
   1:  PR[GP1:91,2] = PR[GP1:90,2] + 4.064;
   1:L PR[91] 10mm/sec CNT100;
   1:  PR[GP1:91,1] = PR[GP1:90,1] + 56.353;
   1:  PR[GP1:91,2] = PR[GP1:90,2] + 8.313;
   1:L PR[91] 10mm/sec CNT100;
   1:  PR[GP1:91,1] = PR[GP1:90,1] + 55.305;
   1:  PR[GP1:91,2] = PR[GP1:90,2] + 13.998;
   1:L PR[91] 10mm/sec CNT100;
   1:  PR[GP1:91,1] = PR[GP1:90,1] + 51.187;
   1:  PR[GP1:91,2] = PR[GP1:90,2] + 20.952;
   1:L PR[91] 10mm/sec CNT100;
   1:  PR[GP1:91,1] = PR[GP1:90,1] + 47.887;
   1:  PR[GP1:91,2] = PR[GP1:90,2] + 26.407;
   1:L PR[91] 10mm/sec CNT100;
   1:  PR[GP1:91,1] = PR[GP1:90,1] + 42.074;
   1:  PR[GP1:91,2] = PR[GP1:90,2] + 31.210;
   1:L PR[91] 10mm/sec CNT100;
   1:  PR[GP1:91,1] = PR[GP1:90,1] + 36.388;
   1:  PR[GP1:91,2] = PR[GP1:90,2] + 35.710;
   1:L PR[91] 10mm/sec CNT100;
   1:  PR[GP1:91,1] = PR[GP1:90,1] + 29.992;
   1:  PR[GP1:91,2] = PR[GP1:90,2] + 38.069;
   1:L PR[91] 10mm/sec CNT100;
   1:  PR[GP1:91,1] = PR[GP1:90,1] + 22.121;
   1:  PR[GP1:91,2] = PR[GP1:90,2] + 40.651;
   1:L PR[91] 10mm/sec CNT100;
   1:  PR[GP1:91,1] = PR[GP1:90,1] + 16.141;
   1:  PR[GP1:91,2] = PR[GP1:90,2] + 40.759;
   1:L PR[91] 10mm/sec CNT100;
   1:  PR[GP1:91,1] = PR[GP1:90,1] + 6.814;
   1:  PR[GP1:91,2] = PR[GP1:90,2] + 40.425;
   1:L PR[91] 10mm/sec CNT100;
   1:  PR[GP1:91,1] = PR[GP1:90,1] + 1.949;
   1:  PR[GP1:91,2] = PR[GP1:90,2] + 38.928;
   1:L PR[91] 10mm/sec CNT100;
   1:  PR[GP1:91,1] = PR[GP1:90,1] + -1.072;
   1:  PR[GP1:91,2] = PR[GP1:90,2] + 39.306;
   1:  PR[GP1:91,3] = PR[GP1:90,3] + 90.440;
   1:L PR[91] 10mm/sec CNT100;
   1:  PR[GP1:91,1] = PR[GP1:90,1] + -5.344;
   1:  PR[GP1:91,2] = PR[GP1:90,2] + 40.618;
   1:L PR[91] 10mm/sec CNT100;
   1:  PR[GP1:91,1] = PR[GP1:90,1] + -15.403;
   1:  PR[GP1:91,2] = PR[GP1:90,2] + 40.979;
   1:L PR[91] 10mm/sec CNT100;
   1:  PR[GP1:91,1] = PR[GP1:90,1] + -20.731;
   1:  PR[GP1:91,2] = PR[GP1:90,2] + 40.882;
   1:L PR[91] 10mm/sec CNT100;
   1:  PR[GP1:91,1] = PR[GP1:90,1] + -29.321;
   1:  PR[GP1:91,2] = PR[GP1:90,2] + 38.065;
   1:L PR[91] 10mm/sec CNT100;
   1:  PR[GP1:91,1] = PR[GP1:90,1] + -35.085;
   1:  PR[GP1:91,2] = PR[GP1:90,2] + 35.937;
   1:L PR[91] 10mm/sec CNT100;
   1:  PR[GP1:91,1] = PR[GP1:90,1] + -41.385;
   1:  PR[GP1:91,2] = PR[GP1:90,2] + 30.952;
   1:L PR[91] 10mm/sec CNT100;
   1:  PR[GP1:91,1] = PR[GP1:90,1] + -46.663;
   1:  PR[GP1:91,2] = PR[GP1:90,2] + 26.595;
   1:L PR[91] 10mm/sec CNT100;
   1:  PR[GP1:91,1] = PR[GP1:90,1] + -50.381;
   1:  PR[GP1:91,2] = PR[GP1:90,2] + 20.446;
   1:L PR[91] 10mm/sec CNT100;
   1:  PR[GP1:91,1] = PR[GP1:90,1] + -54.138;
   1:  PR[GP1:91,2] = PR[GP1:90,2] + 14.089;
   1:L PR[91] 10mm/sec CNT100;
   1:  PR[GP1:91,1] = PR[GP1:90,1] + -55.542;
   1:  PR[GP1:91,2] = PR[GP1:90,2] + 6.344;
   1:L PR[91] 10mm/sec CNT100;
   1:  PR[GP1:91,1] = PR[GP1:90,1] + -56.564;
   1:  PR[GP1:91,2] = PR[GP1:90,2] + 0.002;
   1:L PR[91] 10mm/sec CNT100;
   1:  PR[GP1:91,1] = PR[GP1:90,1] + -56.061;
   1:  PR[GP1:91,2] = PR[GP1:90,2] + -2.764;
   1:L PR[91] 10mm/sec CNT100;
   1:  PR[GP1:91,1] = PR[GP1:90,1] + -55.336;
   1:  PR[GP1:91,2] = PR[GP1:90,2] + -7.603;
   1:L PR[91] 10mm/sec CNT100;
   1:  PR[GP1:91,1] = PR[GP1:90,1] + -54.138;
   1:  PR[GP1:91,2] = PR[GP1:90,2] + -14.099;
   1:L PR[91] 10mm/sec CNT100;
   1:  PR[GP1:91,1] = PR[GP1:90,1] + -50.379;
   1:  PR[GP1:91,2] = PR[GP1:90,2] + -20.458;
   1:L PR[91] 10mm/sec CNT100;
   1:  PR[GP1:91,1] = PR[GP1:90,1] + -46.661;
   1:  PR[GP1:91,2] = PR[GP1:90,2] + -26.607;
   1:L PR[91] 10mm/sec CNT100;
   1:  PR[GP1:91,1] = PR[GP1:90,1] + -41.380;
   1:  PR[GP1:91,2] = PR[GP1:90,2] + -30.963;
   1:L PR[91] 10mm/sec CNT100;
   1:  PR[GP1:91,1] = PR[GP1:90,1] + -35.081;
   1:  PR[GP1:91,2] = PR[GP1:90,2] + -35.949;
   1:L PR[91] 10mm/sec CNT100;
   1:  PR[GP1:91,1] = PR[GP1:90,1] + -29.315;
